	2: 
		WriteFile(
			sNetId := InAmsId,
			hFile := FileHandle,
			pWriteBuff := InPMessage,
			cbWriteLen := InLMessage,
			bExecute := TRUE,
			nErrId => AX_ErrorId[Select],
			bError => AX_Error[Select]
		);
		IF NOT(WriteFile.bBusy) THEN
			IF NOT(WriteFile.bError) THEN
				select := select+1;
				WriteFile(bExecute := FALSE);
				cbWritten := WriteFile.cbWrite;
			ELSE
				select := -1;
			END_IF
		END_IF
	3 : 
		CloseFile(sNetId := InAmsId, 
			hFile := FileHandle,
			bExecute := TRUE, 
			tTimeout := T#1S,
			nErrId => AX_ErrorId[Select],
			bError => AX_Error[Select]
		);
		IF NOT(CloseFile.bBusy) THEN
			IF NOT(CloseFile.bError) THEN
				select := 10;
				CloseFile(bExecute := FALSE);
			ELSE
				select := -1;
			END_IF
		END_IF
		
	10: 
		FileHandle := 0;
		OutBusy := FALSE;
		select := 0;
		OutCompleted := TRUE;
		FOR i := 1 TO NbSteps DO
			AX_ErrorId[i] := 0;
			AX_Error[i] := FALSE;
		END_FOR
		
	-1 : 
		IF FileHandle <> 0 THEN
			CloseFile(sNetId := InAmsId, hFile := FileHandle, bExecute := TRUE);
		END_IF
		OpenFile(bExecute := FALSE);
		WriteFile(bExecute := FALSE);
		IF NOT(CloseFIle.bBusy) THEN
			CloseFile(bExecute := FALSE);
		END_IF
		M_AlarmManager();
		select := 10;
END_CASE

METHOD M_AlarmManager : BOOL
VAR
	j : UINT;
	StringInterm : STRING;
END_VAR
OutError := FALSE;
OutErrorId :='';
FOR j := 1 TO NbSteps DO
	OutError := OutError OR AX_Error[j];
	IF AX_Error[j] THEN
		OutErrorId := concat(concat(Concat(UINT_TO_STRING(j),'_'), UDINT_TO_STRING(AX_ERRORID[j])), CONCAT('*',OutErrorId));
	END_IF
END_FOR
END_METHOD

END_FUNCTION_BLOCK

// ---- 00_FunctionsBlocks/DataProcessing/WriteFile/FUN_CreateDir_CSV.TcPOU
PROGRAM FUN_CreateDir_CSV
VAR_INPUT
	InDirectory 		: T_MaxString;
	Reset2				: BOOL;
END_VAR

VAR
	FB_Time 			: FB_LocalSystemTime;
	MesYear 			: WORD;
	MesMonth			: WORD;
	MesDay				: WORD;
	MesDate				: STRING;
	bTimeOK				: BOOL;
	
	//Dir names 
	CreateDir1			: FB_CreateDir_V2;
	CreateDir2			: FB_CreateDir_V2;
	bFirstDirOk			: BOOL;
	bSecondDirOk		: BOOL;
	bFileOK				: BOOL;
	bDirChange			: BOOL;

END_VAR

VAR_OUTPUT
	
	bInitWrite 			: BOOL;
	AX_DirNames			: ARRAY[1..3] OF t_MaxString; // Folder for years, months and days
	bDirOK				: BOOL;

END_VAR

//	Get time and date  +  Create names
	
IF MesYear <> CalLocalTimeStruct.wYear THEN
	AX_DirNames[1] := Concat(InDirectory, concat(WORD_TO_STRING(CalLocalTimeStruct.wYear), '\'));
	MesYear := CalLocalTimeStruct.wYear;
	bDirChange := TRUE;		
END_IF

IF MesMonth <> CalLocalTimeStruct.wMonth THEN
	AX_DirNames[2] := Concat(AX_DirNames[1], concat(WORD_TO_STRING(CalLocalTimeStruct.wMonth), '\'));
	MesMonth := CalLocalTimeStruct.wMonth;
	bDirChange := TRUE;		
END_IF

IF MesDay <> CalLocalTimeStruct.wDay THEN
	MesDay := CalLocalTimeStruct.wDay;
END_IF		


IF bDirChange OR NOT bFirstDirOk OR NOT bSecondDirOk OR RESET2 THEN
	RESET2 := FALSE;
	bFirstDirOk := FALSE;
	bSecondDirOk := FALSE;
	CreateDir1(InPath := AX_DirNames[1], InExe := TRUE, OutCompleted => bFirstDirOk);
	CreateDir2(InPath := AX_DirNames[2], InExe := bFirstDirOk AND NOT bSecondDirOk, OutCompleted => bSecondDirOk);
	
	IF bFirstDirOk AND bSecondDirOk THEN
		bDirChange := FALSE;
		bDirOK := bFirstDirOk AND bSecondDirOk ;
		CreateDir1(InExe := FALSE);
		CreateDir2(InExe := FALSE);
	END_IF				
END_IF

END_PROGRAM

// ---- 00_FunctionsBlocks/DataProcessing/WriteFile/FB_CreateDir_V2.TcPOU
FUNCTION_BLOCK FB_CreateDir_V2
VAR_INPUT
	InPath 				: T_Maxstring;
	InExe				: BOOL;
END_VAR
VAR_OUTPUT
	OutExiste			: BOOL;
	OutCompleted		: BOOL;
	OutError			: BOOL;
	OutErrorId			: UDINT;
	OutBusy				: BOOL;
END_VAR
VAR
	CreateDir			: FB_CreateDir;	
	
	Trig_Start			: RS;
	Trig				: R_TRIG;
	
	
END_VAR

Trig(CLK := InExe);
//OutCompleted := NOT Trig.Q AND NOT CreateDir.bBusy AND NOT CreateDir.bError;
Trig_Start(SET := Trig.Q);

CreateDir(
	sNetId := '', 
	sPathName := InPath,
	bExecute := Trig.Q
	);
	
IF Trig_Start.Q1 AND NOT CreateDir.bBusy AND (CreateDir.nErrId = 16#723 OR CreateDir.nErrId = 16#70C ) THEN
	createDir(bExecute := FALSE);
	OutExiste := TRUE;
	OutCompleted := TRUE;
	Trig(CLK := FALSE);
	Trig_Start( RESET1 := OutCompleted OR OutError);
	Trig_Start( RESET1 := FALSE);
ELSIF NOT Trig.Q AND Trig_Start.Q1 AND NOT CreateDir.bBusy AND NOT CreateDir.bError THEN
	OutCompleted := TRUE;
	CreateDir(bExecute := FALSE);
	Trig(CLK := FALSE);
	Trig_Start( RESET1 := OutCompleted OR OutError);
	Trig_Start( RESET1 := FALSE);
ELSIF CreateDir.bError THEN
	OutError := TRUE;
	OutErrorId := CreateDir.nErrid;
	CreateDir(bExecute := FALSE);
	Trig(CLK := FALSE);
	Trig_Start( RESET1 := OutCompleted OR OutError);
	Trig_Start( RESET1 := FALSE);

END_IF

OutBusy := Trig_Start.Q1;

END_FUNCTION_BLOCK

// ---- 00_FunctionsBlocks/DataProcessing/ReplaceAll.TcPOU
PROGRAM ReplaceAll
// Replaces all the instances of the input string with another string
// If In_StringToSearch := 'aaaaa123aaaaa123aaaaaaa123aaaaa123'
// In_StringToFind := '123'
// In_StringToReplace : = 'ABC'
// Then : OUT_StringToSearch := 'aaaaaABCaaaaaABCaaaaaaaABCaaaaaABC'
// Equivalent to CTRL + H
VAR_INPUT
	IN_StringToSearch	: T_MaxString;		// String to search : main string with instances we wish to replace
	IN_StringToFind		: STRING;			// String we are looking to find in the String_To_Seach
	IN_StringToReplace 	: STRING;			// String with which we want to replace the String To Find in String To Search
END_VAR

VAR_OUTPUT
	OUT_StringToSearch : T_MaxString;		// Output String
END_VAR

VAR
	KK: INT;
	Test_INT : INT;
END_VAR

OUT_StringToSearch := IN_StringToSearch;
FOR KK := 1 TO LEN(STR := OUT_StringToSearch) DO
	Test_INT := FIND(STR1 := OUT_StringToSearch, STR2 := IN_StringToFind);
	IF Test_INT > 0 THEN
		OUT_StringToSearch := REPLACE(STR1 := OUT_StringToSearch, STR2 := IN_StringToReplace, P := Test_INT, L := len(IN_StringToFind));
		KK := Test_Int;
	END_IF
END_FOR

END_PROGRAM

// ---- 00_FunctionsBlocks/AlarmManagement/FUN_ReadAlarm_CSV.TcPOU
PROGRAM FUN_ReadAlarm_CSV
//Permet de lire les Valeurs de max 1 semaine de points (1 pt/min pdt 7 jours)

VAR_INPUT
	InDirectory_Stockage 		: T_MaxString;		// Base file of the Historization 
	InStartTimeStamp			: TIMESTRUCT;
	InExecute					: BOOL;			//Rising Edge detection of read
	ParamSeparateur				: STRING;
	IN_Reset					: BOOL ; // Close File . 
	ParamMaxLine				: WORD :=  200 ; 
END_VAR                 		

VAR_OUTPUT              		
	OutValue					: ARRAY[1..500] OF ST_ValuesAlarms;
	OutDir						: T_Maxstring;
	OutCompleted				: BOOL;
	OutNbLigne					: UINT;
	OutbBusy					: BOOL;
	OutError 					: BOOL;
	OutErrorID 					: UINT; // 1 : File not found
END_VAR                 		
VAR     
	// Initialisation 
	TypeFile					: STRING;
	ParamTimeOut				: TIME := T#1S;
	
	//Read
	TimeStructBeingRead			: TIMESTRUCT;
	FullDirectory				: STRING;                		
	
	OpenFile					: FB_FileOpen;
	ReadFile					: FB_FileGets;
	CloseFile					: FB_FileClose;
	InfoFile					: FB_EnumFindFileEntry;
	FileInfo					: ST_FindFileEntry;

	Index_Array_OutValue		: UINT := 1;			// Valeur de OutValue qui va être écrite
	
	Opening						: BOOL := TRUE;
	
	LineRead					: T_Maxstring;
	EOF_Reached					: BOOL;              		
	CompteurLigne				: CTU;
	AX_ArrayString 				: ARRAY[1..100] OF T_Maxstring;
	
	OutEmpty					: ARRAY[1..500] OF ST_ValuesAlarms;
	OutBusy						: RS;
	OutCompleted_RS				: RS;
	Trig_Read					: R_TRIG;
	Trig_Start 					: R_TRIG;
	
	FileHandle					: UINT;
	FileHandle_Old				: UINT;
	
	KK: UINT := 1;
	bInit : BOOL;
	LL: UINT;
	MM: UINT;
END_VAR

Trig_Start(CLK := InExecute);
OutCompleted_RS(Reset1 := Trig_Start.Q);
IF trig_start.Q THEN
	OutEmpty := OutValue;
	outError := FALSE;
END_IF
OutBusy(Set := InExecute, RESET1 := OutError OR OutCompleted_RS.Q1);
OutbBusy := OutBusy.Q1;
OutCompleted := OutCompleted_RS.Q1;
IF OutBusy.Q1 THEN	
	// J'initialise le tout : 
	//Initialisation du type de fichier
	TypeFile := 'ALARMS'; 
	
	TimeStructBeingRead := DT_TO_SYSTEMTIME(SYSTEMTIME_TO_DT(InStartTimeStamp) );
	FullDirectory := Concat(Concat(Concat(Concat(Concat(Concat(Concat(Concat(Concat(Concat(Concat(Concat(InDirectory_Stockage , WORD_TO_STRING(TimeStructBeingRead.wyear)),'\'),WORD_TO_STRING(TimeStructBeingRead.wMonth)),'\'),'ALARMS'),'_'),WORD_TO_STRING(TimeStructBeingRead.wyear)),'-'),WORD_TO_STRING(TimeStructBeingRead.wMonth)),'-'),WORD_TO_STRING(TimeStructBeingRead.wDay)),'.csv');
    OutDir := FullDirectory;
	//Ouverture du Fichier, récupération du handle
	OpenFile
	(
		sNetId := '',
		sPathName := FullDirectory,
		nMode := FOPEN_MODEREAD,
		ePath := PATH_GENERIC,
		bExecute := Opening AND NOT OutCompleted_RS.Q1,
		hFile => FileHandle
	);
	
	IF OpenFile.nErrId = 1804 THEN // Le fichier n'existe pas 
		OutErrorID := 1;
		OutError := OpenFile.bError;
		OpenFile(bExecute :=  FALSE);
	ELSIF OpenFile.bError THEN		// Il y a eu une autre erreur
		OutError := OpenFile.bError;
	ELSIF NOT OpenFile.bError AND NOT OpenFile.bBusy AND FileHandle <> 0 AND FileHandle <> FileHandle_Old THEN
		opening := FALSE;
		FileHandle_Old := FileHandle;
	END_IF
	// On a obtenu le file handle, on va commencer la lecture

	// Le bloc suivant va lire le document ligne à ligne en incrémentant le compteur ligne et en ressortant l'ensemble de la ligne dans LineRead
	LineRead := '';
	IF NOT opening THEN
		ReadFile
		(
			sNetId := '',
			hFile := FileHandle,
			bExecute := TRUE,
			tTimeout := ParamTimeOut,
			sLine => LineRead,
			bEOF => EOF_Reached
		);				

		IF NOT ReadFile.bBusy AND NOT ReadFile.bError AND (LineRead <> '') THEN
			ReadFile(bExecute := FALSE);
			CompteurLigne(CU := TRUE);	
			CompteurLigne(CU := FALSE);
			IF CompteurLigne.CV > 2 THEN
				Split(IN_TextToSearch := LineRead, IN_Delimiter := 	ParamSeparateur, OUT_Split => AX_ArrayString);			
				OutValue[Index_Array_OutValue].TimeStamp_Act 	:= AX_ArrayString[1];
				OutValue[Index_Array_OutValue].ID 				:= STRING_TO_UINT(AX_ArrayString[2]);
				OutValue[Index_Array_OutValue].Message			:= AX_ArrayString[3];
				OutValue[Index_Array_OutValue].Value			:= STRING_TO_BOOL(AX_ArrayString[4]);
				OutValue[Index_Array_OutValue].Ack			 	:= STRING_TO_BOOL(AX_ArrayString[5]);
				OutValue[Index_Array_OutValue].Alarms_LVL	 	:= STRING_TO_UINT(AX_ArrayString[6]);				
				Index_Array_OutValue := Index_Array_OutValue + 1;
				
			END_IF
		
		ELSIF NOT ReadFile.bBusy AND  ReadFile.bError THEN
			OutError := TRUE;	
		ELSIF  EOF_Reached THEN
			OutNbLigne := Index_Array_OutValue;
			OutCompleted_RS( SET := TRUE);
			OutCompleted_RS( SET := FALSE);
	
		END_IF	
	
	END_IF
	
ELSIF EOF_Reached AND FileHandle <> 0 THEN
	ReadFile(bExecute := FALSE);
	CloseFile
	(
		sNetId := '',
		bExecute := TRUE,
		hFile := FileHandle,
		tTimeout := ParamTimeOut
	);
	IF NOT CloseFile.bBusy AND NOT CloseFile.bError THEN
		CloseFile(bExecute := FALSE);
		Opening := TRUE;
		CompteurLigne(RESET := TRUE);
		CompteurLigne(RESET := FALSE);
		Index_Array_OutValue := 1;
		FileHandle := 0;
		OutValue := OutEmpty;
	ELSIF NOT CloseFile.bBusy AND closefile.bError THEN
		OutError := TRUE;
	END_IF  
END_IF

END_PROGRAM

// ---- 00_FunctionsBlocks/DataProcessing/Split.TcPOU
PROGRAM Split
//Donne la position de la IN_Position-ième répétition du caractère recherché et renvoie la chaine de caractère suivante
VAR_INPUT
	IN_Delimiter 		: STRING;
	IN_TextToSearch		: T_MaxString;
END_VAR

VAR
	n					: UINT;	
	Position_Int		: UINT;
	LenOutSplit			: INT;
	TextToSearch_Int	: T_MaxString;
	OUT_Null			: ARRAY[1..100] OF T_Maxstring;
END_VAR

VAR_OUTPUT
	OUT_Split			: ARRAY[1..100] OF T_Maxstring;
	NbElements			: UINT;
END_VAR

OUT_Split := OUT_Null;
n:= 1;
TextToSearch_Int := IN_TextToSearch;
Position_Int := INT_TO_UINT( Find(STR1 := TextToSearch_Int, STR2 := IN_Delimiter));
LenOutSplit := 0;

WHILE Position_Int > 0 AND LenOutSplit < LEN(STR:= IN_TextToSearch) DO
	OUT_Split[n] := LEFT(STR := TextToSearch_Int, SIZE := UINT_TO_INT(Position_Int)-1);
	LenOutSplit := LenOutSplit + Len(STR := OUT_Split[n])+1;
	TextToSearch_Int := RIGHT(STR := TextToSearch_Int, SIZE := LEN(STR:= TextToSearch_Int)- LEN(STR:= OUT_Split[n])-1);
	Position_Int := INT_TO_UINT(FIND(STR1 := TextToSearch_Int, STR2 := IN_Delimiter));
	n := n + 1;
END_WHILE

NbElements := n-1;

END_PROGRAM

// ---- 00_FunctionsBlocks/AlarmManagement/SMS_Server.TcPOU
PROGRAM SMS_Server
VAR PERSISTENT
	AX_Numtel						: ARRAY[1..CstNbUser] OF STRING(26) ;	//Contient tous les numéros des utilisateurs
	AX_Subscribed					: ARRAY[1..CstNbUser] OF BOOL ;			//Contient tous les états d'abonnements des utilisateurs aux SMS
	AX_NomUtili						: ARRAY[1..CstNbUser] OF STRING(50);	//Contient tous les noms des utilisateurs
	AX_User_LVL						: ARRAY[1..CstNbUser] OF WORD;			//Contient tous les niveau d'adhésion des utilisateurs.
END_VAR

VAR_INPUT
	IN_DataSetFifo_ReadSMS			: FB_SMSDatasetFifo_Read; //Buffer automate des sms récuperer depuis modem Gsm
	IN_DataSetFifo_SendSMS			: FB_SMSDatasetFifo_Send; //Buffer automate des sms récuperer depuis modem Gsm	
	IN_AX_Journal					: ARRAY [0..CstNbAlarmCode] OF ARRAY[0..15] OF ST_ValuesAlarms; //Journal d'envoi, contient destinataire et message, et gestion de l'envois ou pas du sms
	IN_Reset_OPC					: BOOL;
	IN_ChangePhoneMailInfos_OPC			: BOOL;
	IN_Reset_SmsServer				: BOOL;
	IN_CmdReset_L					: BOOL;
	IN_CmdDeleteAllSms			: BOOL;
END_VAR

VAR
	fbSerialLineControl		: SerialLineControl;
	stTxBufferPC			: ComBuffer;
	stRxBufferPC			: ComBuffer;
	fbReadSMS				: FB_ReadSMS;
	fbSendSMS				: FB_SendSMS;
	fbDeleteSMS				: FB_DeleteSMS;
	fbDeleteAllSMS			: FB_DeleteAllSMS;
	Fblogin 				: FB_Login;
	
	//READ VARIABLE 
	bStartRead				: BOOL; //Gestion du front montant FB ReadSMS
	ReadSMS_bBusy			: BOOL;
	ReadSMS_bError			: BOOL;
	ReadSMS_nErrorID		: UINT;
	
	LoginSMS_bError			: BOOL;
	LoginSMS_bBusy		    : BOOL;
	IndexReadMessage		: USINT:=1; //Index du message a lire
	ReadSMS_MessageText		: STRING(240); // Message brut du SMS recu
	Etape_Read 		 		: SINT:=0; // Etape du Case de M_Fill_Buffer_Read
	Message_Tous_lu 		: BOOL;  // Si tous les message du buffer READ sont lu : True sinon False
	
	//DELETE VARIABLE
	bStartDelete			: BOOL; //Gestion du front montant FB DeleteSms
	DeletedSMS_bBusy		: BOOL;
	DeletedSMS_Error		: BOOL;
	DeletedSMS_nErrorID		: UINT;
	
	IndexDeleteMessage 		: USINT:=1; //Index du message a supprimer
	
	//SEND VARIABLE
	bStartSend				: BOOL;
	Message_Send			: STRING(160);
	MesTimeStamp			: STRING(17);
	SendSMS_bBusy			: BOOL;
	SendSMS_bError			: BOOL;
	Etape_Send				: SINT;
	CPT						: SINT:=1;
	Num_Tel					: STRING(30);

	//INIT VARIABLE
	bStartlogin             : BOOL:=TRUE; //Gestion du front montant FB login
	bInit					: BOOL;
	
	//Variables de All Delete
	DeletedAllSMS_bBusy		: BOOL;
	DeletedAllSMS_Error		: BOOL;
	DeletedAllSMS_nErrorID	: UINT;
	G7_DelAll				: SINT;

	Bstart_delete_all		: BOOL;    
	
	//M_G7_SMS
	CPT_Message				: CTU;
	


	//TABLEAU
	AX_MesAlarmCode_Bool	: ARRAY [1..CstNbAlarmCode] OF ARRAY[1..15] OF BOOL; //Tableau de tous les alarmesCode en Bool
	AX_Alarm_State			: ARRAY [1..CstNbAlarmCode] OF ARRAY[1..15] OF BOOL; //Tableau de Bool avec toutes les nouveaux bit modifiés
	fbXorWord				: FB_XorWord; //Compare 2 Word et retourne les bit modifié
	Extract_Num_Mes			: FB_Extract_Num_Mes; //Extraction des infos: Message,Numero de tel

	// M_Evaluate
	MesDataExd.MesData			: ServerSMS;
	CalNbrUtiliActive    : INT := 10;
	//AlarmCode
	RS_LoginSMS_bError		: RS;
	RS_SendSMS_bError       : RS;
	RS_ReadSMS_bError       : RS;
	RS_DeletedSMS_Error     : RS;
    RS_DeletedAllSMS_Error  : RS;

	AX_Cmd_SMS				: ARRAY[1..CstNbCMD] OF STRING(26):=['Infos','Reboot_ADSL','P_Onduleur','Stop_SMS','Start_SMS','Toggle subscription','Ip Publique','Active Alarms','Help','Test SMS','ForcedStayConnect','Restart HHCollector','Restart PLC','Auto Couplage','Disconnect', 'VPN Connect', 'VPN Disconnect', 'Reboot_IPC']; //Contient toutes les commandes possibles

	Serial_Use				: BOOL:=TRUE;
	ReadAct					: BOOL:=FALSE;
	LoginOK                 : BOOL:=TRUE;
	Reset					: BOOL;
	
	//OPC
	RS_OPC					: RS;
	RS_Deletteall			: RS;
	RS_Reset				: RS;
	Trig_OPC				: R_TRIG;
	Trig_OpcDelAll			: R_TRIG;
	Trig_OpcReset			: R_TRIG;

	
	
END_VAR

IF NOT bInit THEN
	M_Init();
ELSE
	
	// READ OPC Data .
	M_OPC();

	//SERIALLINEMODE_EL6_22B	
	fbSerialLineControl(Mode:= SERIALLINEMODE_PC_COM_PORT ,
		pComIn:= ADR(stPCComInData),
		pComOut:= ADR(stPCComOutData),
		SizeComIn:= UINT_TO_INT( SIZEOF(stPCComInData)),
		TxBuffer:= stTxBufferPC,
		RxBuffer:= stRxBufferPC,
		Error=> ,
		ErrorID=> );
		
	Fblogin(bStart:=bStartlogin ,					// etrangement le login fonctionne puis fait une erreur , puis refonctionne etc . relance du login sur read error je pense qui entraine une tentative de login qui foire. 	
			stTxBuffer:=stTxBufferPC,	
			stRxBuffer:=stRxBufferPC,
			bBusy =>LoginSMS_bBusy,
			bError=>LoginSMS_bError
			);		
		
	fbSendSMS(bStart:= bStartSend,
		sPhoneNumber:= Num_Tel,
		bReset := IN_Reset_OPC ,
		sSMSText:= Message_Send,
		stTxBuffer:=stTxBufferPC ,
		stRxBuffer:=stRxBufferPC,
		bBusy=>SendSMS_bBusy,
		bError=>SendSMS_bError);
	
	fbReadSMS(bStart:= bStartRead,
		nIndex:= IndexReadMessage,
		stTxBuffer:=stTxBufferPC ,
		stRxBuffer:=stRxBufferPC ,
		bBusy=> ReadSMS_bBusy,
		bError=> ReadSMS_bError,
		nErrorID=> ReadSMS_nErrorID
		);
	
	
	fbDeleteSMS
	(
		bStart:= bStartDelete,
		nIndex:= IndexDeleteMessage,
		stTxBuffer:=stTxBufferPC,
		stRxBuffer:=stRxBufferPC,
		bBusy=> DeletedSMS_bBusy,
		bError=> DeletedSMS_Error,
		nErrorID=> DeletedSMS_nErrorID
	);
	
	fbDeleteAllSMS
	(
		bStart:= Bstart_delete_all,
		stTxBuffer:=stTxBufferPC,
		stRxBuffer:=stRxBufferPC,
		bBusy=> DeletedAllSMS_bBusy,
		bError=> DeletedAllSMS_Error,
		nErrorID=> DeletedAllSMS_nErrorID
	);	

	M_DeleteAll();
	M_Fill_Buffer_Read(); //Lecture de tous les messages recu

	M_AlarmManager();
	M_Evaluate();		// Update serveur info
	M_Send(); // Envois de tous les messages (Alarm ou réponce aux sms de cmd)

	M_Cmd_Execute(); // Verification des messages recu
	
	IF Reset OR IN_Reset_OPC  THEN
		M_Reset();
	END_IF
	
	IF NOT LoginSMS_bBusy AND NOT LoginSMS_bError AND LoginOK THEN
		BstartLogin := FALSE;
		Serial_Use:=FALSE;
		LoginOK:=FALSE;
	END_IF
	
	
END_IF

METHOD M_AlarmManager
VAR
	ii:SINT;
	jj:INT;
	KK:INT;
	FB_AlarmCodeManager			: FB_AlarmCodeManager ;
END_VAR
RS_LoginSMS_bError(SET:=LoginSMS_bError,RESET1:=	IN_CmdReset_L OR IN_Reset_OPC); 		
RS_SendSMS_bError(SET:=SendSMS_bError,RESET1:=  	IN_CmdReset_L OR IN_Reset_OPC); 		
RS_ReadSMS_bError(SET:=ReadSMS_bError,RESET1:=  	IN_CmdReset_L OR IN_Reset_OPC); 		
RS_DeletedSMS_Error(SET:=DeletedSMS_Error,RESET1:=	IN_CmdReset_L OR IN_Reset_OPC); 		
RS_DeletedAllSMS_Error(SET:=DeletedAllSMS_Error,RESET1:=IN_CmdReset_L OR IN_Reset_OPC); 	

// ALARM CODE //
	FB_AlarmCodeManager(
		bAlarm1			:= RS_LoginSMS_bErrOR.Q1		  ,			// Login SMS Error
		bAlarm2			:= RS_SendSMS_bErrOR.Q1		   ,			// Send SMS Error
		bAlarm3			:= RS_ReadSMS_bErrOR.Q1		   ,			// Read SMS Error 
		bAlarm4			:= RS_DeletedSMS_ErrOR.Q1		 ,			// Delete SMS Error 
		bAlarm5			:= RS_DeletedAllSMS_ErrOR.Q1	,			// Delete All Sms Error
		bAlarm6			:= IN_DataSetFifo_ReadSMS.bOverwrite,		// Read Fifo overflow
		bAlarm7			:= IN_DataSetFifo_SendSMS.bOverwrite,       // Send Fifo overflow
		bAlarm8			:= FALSE,                                   //
		bAlarm9			:= FALSE,                                   //
		bAlarm10		:= FALSE,                                   //
		bAlarm11		:= FALSE,									//
		bAlarm12		:= FALSE,                                   //
		bAlarm13		:= FALSE,                                   //
		bAlarm14		:= FALSE,                                   //
		bAlarm15		:= FALSE,                                   //
		wAlarmCode		=>MesData.MesAlarmCode);
END_METHOD

METHOD M_Cmd_Execute
VAR_INPUT
END_VAR

VAR
	i: SINT;
	Num_Valide 		: BOOL;
	Message_Valide 	: BOOL;
	Index_CMD 		: SINT;
END_VAR
IF IN_DataSetFifo_ReadSMS.nCount > 0 THEN
	IN_DataSetFifo_ReadSMS.A_Get(); // Récuperation du FIFO
	FOR i:=1 TO CstNbUser DO // VERIFICATION du numéro de telephone
		IF AX_Numtel[i]=IN_DataSetFifo_ReadSMS.Out.Num THEN
			Num_Valide := TRUE;
			EXIT;
		END_IF
	END_FOR
	IF Num_Valide THEN
		FOR i:=1 TO CstNbCMD DO // VERIFICATION du message
			IF IN_DataSetFifo_ReadSMS.Out.Message=AX_Cmd_SMS[i] THEN
				Message_Valide := TRUE;
				Index_CMD:=i;
				EXIT;
			END_IF
		END_FOR
	END_IF
	
	IF Num_Valide AND Message_Valide THEN
		M_G7_SMS(G7_Etape:=Index_CMD);

	ELSE
		IN_DataSetFifo_ReadSMS.A_Remove(); //IL s'agit d'un spam ou d'un utilisateur non autorisé
	END_IF
	

END_IF
END_METHOD

METHOD M_DeleteAll


VAR
	
END_VAR
CASE G7_DelAll OF
	
	0: // Entrée
		IF RS_Deletteall.Q1 AND NOT Serial_Use THEN
			Serial_Use 			:= TRUE;
			Bstart_delete_all 	:= TRUE;
			G7_DelAll 			:= 1;
		END_IF
	1: // attente du bb=usy
		Bstart_delete_all 	:= FALSE;
		IF NOT DeletedAllSMS_bBusy OR DeletedAllSMS_Error THEN
			RS_Deletteall(RESET1:= TRUE);
			RS_Deletteall(RESET1:= FALSE);
			Serial_Use 			:= FALSE;
			G7_DelAll 			:= 0;
		END_IF
		
		
END_CASE
END_METHOD

METHOD M_Evaluate
VAR 
	KK: INT;
END_VAR
CalNbrUtiliActive := 0 ;
FOR KK:=1 TO CstNbUser DO 
	IF 	AX_Numtel[KK] <> '' THEN 
		CalNbrUtiliActive := CalNbrUtiliActive+1 ; 
	END_IF
END_FOR



Mesdata.NbrUtiliActive 	:= CalNbrUtiliActive ;
Mesdata.AX_Numtel		:= AX_Numtel			;
Mesdata.AX_Subscribed	:= AX_subscribed	    ;
MesData.AX_NomUtili		:= AX_NomUtili		    ;
MesData.AX_UserLVL		:= AX_User_LVL		    ;
END_METHOD

METHOD M_Fill_Buffer_Read
CASE Etape_Read OF
	0://Initilisation
		IF NOT ReadSMS_bBusy AND NOT Serial_Use AND ReadAct THEN
			Etape_Read:=10;
			ReadSMS_MessageText:='';
			bStartlogin:=TRUE;
			Serial_Use:=TRUE;
		END_IF
	10: //Initialisation MODEM (ECHO OFF)
		//Serial_Use:=TRUE;
		bStartlogin:=FALSE;
		IF NOT LoginSMS_bBusy AND NOT LoginSMS_bError THEN
			Etape_Read:=1;
			BstartRead:=TRUE;	
		ELSIF LoginSMS_bError THEN
			Etape_Read:=0;
			Serial_Use:=FALSE;
		END_IF
	1://Lecture des sms
		//GVL_Rapale.Serial_Use:=TRUE;
		ReadSMS_MessageText:=fbReadSMS.sMessageText;
		BstartRead:=FALSE;	
		IF NOT ReadSMS_bBusy AND NOT ReadSMS_bError THEN	
			Etape_Read:=2;
			Serial_Use:=FALSE;
		ELSIF ReadSMS_bError THEN
			Etape_Read:=0;
			Serial_Use:=FALSE;
			
		END_IF
		
	2://Analyse du sms en Cas d'un message non vide
		IF(ReadSMS_MessageText<>'OK$R$N') AND (ReadSMS_MessageText<>'') THEN
			
			IF (FIND(ReadSMS_MessageText,'REC UNREAD')>0) THEN		//
				Message_Tous_lu := FALSE;
				IndexReadMessage:=IndexReadMessage+1;
				Extract_Num_Mes(InMessage:=ReadSMS_MessageText);
				IN_DataSetFifo_ReadSMS.A_Add( in := Extract_Num_Mes.OutDataEntry);
				Etape_Read:=0;					
			ELSE	// Messages have already been read. 
				Message_Tous_lu := TRUE;
				IndexReadMessage:=IndexReadMessage+1;
				ReadSMS_MessageText:='';
				Etape_Read:=0;
			END_IF
		ELSE
			Etape_Read:=3;
		END_IF
	3://Analyse du sms en cas de message vide
		IF Message_Tous_lu THEN
			Etape_Read:=4;
		ELSE
			IndexReadMessage:=1;
			Etape_Read:=0;
		END_IF
	4://Initialisation du Delete_FB
		IF NOT DeletedSMS_bBusy AND ReadAct THEN //AND NOT GVL_Rapale.Serial_Use THEN
			Etape_Read:=5;
			bStartDelete:=TRUE;
			Serial_Use:=TRUE;
		END_IF
	5://Suppression du buffer GSM
		//GVL_Rapale.Serial_Use:=TRUE;
			bStartDelete:=FALSE;
		IF NOT DeletedSMS_bBusy AND NOT DeletedSMS_Error THEN
			Serial_Use:=FALSE;
			Etape_Read:=6;
		ELSIF DeletedSMS_Error THEN
			//GVL_Rapale.Serial_Use:=FALSE;
			Etape_Read:=4;
			Serial_Use:=FALSE;
		END_IF
	6://Controle suppression
		IF IndexDeleteMessage=IndexReadMessage-1 THEN
			Etape_Read:=0;
			IndexDeleteMessage:=1;
			Message_Tous_lu:=FALSE;
			IndexReadMessage:=IndexReadMessage+1;
			Serial_Use:=FALSE;
		ELSE
			IndexDeleteMessage:=IndexDeleteMessage+1;
			Etape_Read:=4;
		END_IF		
		
END_CASE
END_METHOD

METHOD M_G7_SMS
VAR_INPUT
	G7_Etape :SINT;
END_VAR

VAR
	InStruct 		: ST_ValuesAlarms;
END_VAR
FUN_Alarms.M_G7_SMS(
	DataSetFifo_ReadSMS		:= IN_DataSetFifo_ReadSMS,
    IN_DataSetFifo_SendSMS	:= IN_DataSetFifo_SendSMS,
 	CPT_Message				:= CPT_Message,	
    InStruct 				:= InStruct,
    G7_Etape 				:= G7_Etape,
    AX_Numtel				:= AX_Numtel,
    AX_subscribed			:= AX_subscribed,
    AX_MesAlarmCode_Bool	:= AX_MesAlarmCode_Bool,
    AX_Cmd_SMS		        := AX_Cmd_SMS
);
END_METHOD

METHOD M_Init

//Initialisation BUFFER

	//Buffer pour la lecture des sms
	IN_DataSetFifo_ReadSMS.A_Reset();
	IN_DataSetFifo_ReadSMS.A_Add();
	IN_DataSetFifo_ReadSMS.A_Get();
	IN_DataSetFifo_ReadSMS.A_Remove();
	
	//Buffer pour l'envois des sms
	IN_DataSetFifo_SendSMS.A_Reset();
	IN_DataSetFifo_SendSMS.A_Add();
	IN_DataSetFifo_SendSMS.A_Get();
	IN_DataSetFifo_SendSMS.A_Remove();

//Initialisation du Journal		
bInit := TRUE;
END_METHOD

METHOD M_OPC : BOOL
VAR
	AX_Numtel_Init				: ARRAY[1..CstNbUser] OF STRING(26);
END_VAR
Trig_OPC(CLK := IN_ChangePhoneMailInfos_OPC);
Trig_OpcDelAll(CLK := IN_CmdDeleteAllSms);
Trig_OpcReset(CLK:= IN_Reset_SmsServer);

RS_OPC(SET:= Trig_OPC.Q);
RS_Deletteall(SET:=Trig_OpcDelAll.Q);
RS_Reset(Set:=Trig_OpcReset.Q);

IF (*NOT Serial_Use AND*) RS_OPC.Q1 THEN
	//Numéro de téléphone
	AX_Numtel := OpcUa.AllValueW.AX_NbPhone_OPC;
	//Nom d'utilisateur
	AX_NomUtili	:= OpcUa.AllValueW.AX_NamesUsers_OPC;
	
	// User LVL . 
	AX_User_LVL := OpcUa.AllValueW.AX_UserLVL;

	//Gestion subscription
	AX_Subscribed := OpcUa.AllValueW.AX_SubscribedSms_OPC;

	RS_OPC(RESET1:= TRUE);
	RS_OPC(Reset1 := FALSE);
END_IF

IF RS_Reset.Q1 THEN
	IN_Reset_Opc := TRUE;
END_IF
END_METHOD

METHOD M_Reset : BOOL
VAR_INPUT
END_VAR
IN_DataSetFifo_SendSMS.A_Reset();

bStartRead 		:= FALSE;
bStartSend 		:= FALSE;
bStartDelete 	:= FALSE;
bStartlogin 	:= FALSE;
Serial_Use		:= FALSE;


SendSMS_Berror := FALSE ;
ReadSMS_bError := FALSE ;
LoginSMS_bError := FALSE ; 
DeletedSMS_Error := FALSE ; 
DeletedAllSMS_Error := FALSE ; 

RS_Reset(RESET1 := TRUE);
RS_Reset(RESET1 := FALSE);
Reset 			:= FALSE;
IN_Reset_OPC 		:= FALSE;
END_METHOD

METHOD M_Send
VAR_INPUT
END_VAR

CASE ETAPE_Send OF
	0://Etape d'entree
		IF NOT SendSMS_bBusy  AND NOT Serial_Use AND IN_DataSetFifo_SendSMS.nCount > 0 AND NOT LoginSMS_bBusy AND NOT LoginSMS_bError THEN  //Si serial libre et buffer contient plus d'une infos
			ReadAct:=FALSE;	
			Serial_Use:=TRUE;
			//bStartSend:=TRUE;
			SendSMS_bError := FALSE;
			Num_Tel := '';
			Message_Send:='';
			IN_DataSetFifo_SendSMS.A_Get();  //recuperation du message dans le send buffer 
			ETAPE_Send := 20  ; 
		ELSE
			ReadAct:=TRUE;	// En attente de lecture de mot d'alarme
		END_IF
			
		20:// Check les utilisateurs pour l'envoi des SMS 
			IF AX_Numtel[CPT] <> '' AND  AX_Subscribed[CPT] AND IN_DataSetFifo_SendSMS.out.Num_tel = '' AND (AX_User_LVL[CPT] AND IN_DataSetFifo_SendSMS.out.Alarms_LVL)>0    THEN
				// On envoi l'alarme si l'utilisateur est subscribed , et est dans la liste de diffusion de l'alarme
				Num_Tel:=AX_NumTel[CPT];
				bStartSend:=TRUE;
				ETAPE_Send:=1;
				MesTimeStamp := CONCAT(REPLACE(STR1:= IN_DataSetFifo_SendSMS.Out.TimeStamp_Act, STR2 := ' ', L := 1, P := 11), ' ') ;

				Message_Send := CONCAT(str1:=CONCAT(str1:=CONCAT(str1:=MesTimeStamp, str2:='$NID:' ), STR2:= UINT_TO_STRING(IN_DataSetFifo_SendSMS.out.ID)), STR2:=' ,' ) ; 
				Message_Send := CONCAT(STR1:=Message_Send , STR2:= IN_AX_Journal[IN_DataSetFifo_SendSMS.out.IndexWord][IN_DataSetFifo_SendSMS.Out.IndexBit].Message);
				
				IF IN_DataSetFifo_SendSMS.OUT.Active  THEN //Connaitre le statut de l'alarme: Active ou Non active
					Message_Send:=Concat(left(Message_Send, 125),' : Active');	// ajout de la mention activee ou desactive 
				ELSE
					Message_Send:=concat(left(Message_Send, 125),' : Desactive');
				END_IF
			ELSIF ( NOT AX_Subscribed[CPT] OR (AX_User_LVL[CPT] AND IN_DataSetFifo_SendSMS.out.Alarms_LVL)=0  ) AND IN_DataSetFifo_SendSMS.out.Num_tel = ''  THEN
				// L'alarme n'est pas envoyéeà cet utilisateur	
				Num_Tel := '';
				ETAPE_Send:=2;
			ELSIF IN_DataSetFifo_SendSMS.out.Num_tel <> ''  THEN
				// Si un numero de telephone est renseigné précisement, on envoi à ce numéro quelque soit la liste de diffusion , ou si l'utilisateur est subscribed
				bStartSend:=TRUE;
				Message_Send := CONCAT(STR1:=Message_Send , STR2:= IN_AX_Journal[IN_DataSetFifo_SendSMS.out.IndexWord][IN_DataSetFifo_SendSMS.Out.IndexBit].Message);
				Num_Tel:=IN_DataSetFifo_SendSMS.Out.Num_tel;
				ETAPE_Send:=1;
			ELSE
				// L'alarme n'est pas envoyée		
				Num_Tel := '';
				ETAPE_Send:=2;
			END_IF

	1://Envois du message
		Bstartsend:=FALSE;	
		IF NOT SendSMS_bBusy  THEN
			IF IN_DataSetFifo_SendSMS.OUT.IndexWord > 0 AND IN_DataSetFifo_SendSMS.In.Num_tel = ''   THEN
				ETAPE_Send:=2; // Alarme
				
			ELSE
				ETAPE_Send:=3; // Retour Sms ou utilisateur de renseignée
			END_IF
		ELSIF NOT SendSMS_bBusy AND SendSMS_Berror THEN // GGY
			//ETAPE_Send:=0; modif lWN seminaire 26/08/2020, gestion des ATE0, si erreur on supprime tout de meme le sms.
			ETAPE_Send:= 3;
			SendSMS_Berror := FALSE ; // On reset l'error apres avoir supprimé le SMS . 
			
		END_IF
		
	2:// Switch a un autre utilisateur
		IF CPT< CstNbUser THEN
			CPT:=CPT+1;
			ETAPE_Send:=20;
		ELSE
			ETAPE_Send:=3;
		END_IF
	
	3://Suppression de l'alarme et on passe au prochaine element dans le fifo
		IN_DataSetFifo_SendSMS.A_Remove();
		CPT:=1;
		Message_Send:='';
		ETAPE_Send:=0;
		Serial_Use:=FALSE;
		bStartSend:=FALSE;

END_CASE
END_METHOD

END_PROGRAM

// ---- 00_FunctionsBlocks/Fifo/FB_SMSDatasetFifo_Read.TcPOU
FUNCTION_BLOCK FB_SMSDatasetFifo_Read
VAR_INPUT
    bOverwrite : BOOL;
    In         : ST_SMSDataSetEntry_Read;
END_VAR
VAR_OUTPUT
    bOk        : BOOL;
    nCount     : UDINT;
    nLoad      : UDINT;
    Out        : ST_SMSDataSetEntry_Read;
END_VAR
VAR
    arrBuffer  : ARRAY[0..Max_buffer_size_G] OF BYTE; (* Buffer memory used by FB_MemRingBuffer function block *)
    fbBuffer   : FB_MemRingBuffer;
END_VAR

ACTION A_Add:
fbBuffer.A_AddTail(pWrite := ADR(in),
						   cbWrite:=SIZEOF(in),
						   pBuffer:=ADR(arrBuffer),
						   cbBuffer:=SIZEOF(arrBuffer),
						   bOK=>bOK,
						   nCount =>nCount);
IF NOT bOK THEN 
	IF bOverwrite THEN
		fbBuffer.A_RemoveHead();(*remove one oldest entry*)
		fbBuffer.A_AddTail(bOK => bOk,nCount => nCount);
	END_IF
END_IF

nload := (fbbuffer.cbSize * 100)/(Max_buffer_size_G);
END_ACTION

ACTION A_Get:
fbBuffer.A_GetHead(pWrite := ADR(out),
						   cbWrite:=SIZEOF(out),
						   pBuffer:=ADR(arrBuffer),
						   cbBuffer:=SIZEOF(arrBuffer),
						   bOK=>bOK,
						   nCount =>nCount);
nload := (fbbuffer.cbSize * 100)/(Max_buffer_size_G);
END_ACTION

ACTION A_Remove:
fbBuffer.A_RemoveHead(pRead:=ADR(out),
						cbRead:=SIZEOF(out),
						pBuffer:=ADR(arrBuffer),
						cbBuffer:=SIZEOF(arrBuffer),
						bOK=>bOK,
						nCount =>nCount);
nload := (fbbuffer.cbSize * 100)/(Max_buffer_size_G);
END_ACTION

ACTION A_Reset:
MEMSET(ADR(arrBuffer),0,SIZEOF(arrBuffer)); (*reset internal buffer*)
fbBuffer.A_Reset(bOK=>bOK,nCount=>ncount);
nload := (fbbuffer.cbSize * 100)/(Max_buffer_size_G);
END_ACTION

END_FUNCTION_BLOCK

// ---- 00_FunctionsBlocks/Fifo/FB_SMSDatasetFifo_Send.TcPOU
FUNCTION_BLOCK FB_SMSDatasetFifo_Send
VAR_INPUT
    bOverwrite : BOOL;
    In         : ST_SMSDataSetEntry_Send;
END_VAR
VAR_OUTPUT
    bOk        : BOOL;
    nCount     : UDINT;
    nLoad      : UDINT;
    Out        : ST_SMSDataSetEntry_Send;
END_VAR
VAR
    arrBuffer  : ARRAY[0..Max_buffer_size_G] OF BYTE; (* Buffer memory used by FB_MemRingBuffer function block *)
    fbBuffer   : FB_MemRingBuffer;
END_VAR

ACTION A_Add:
fbBuffer.A_AddTail(pWrite := ADR(in),
						   cbWrite:=SIZEOF(in),
						   pBuffer:=ADR(arrBuffer),
						   cbBuffer:=SIZEOF(arrBuffer),
						   bOK=>bOK,
						   nCount =>nCount);
IF NOT bOK THEN 
	IF bOverwrite THEN
		fbBuffer.A_RemoveHead();(*remove one oldest entry*)
		fbBuffer.A_AddTail(bOK => bOk,nCount => nCount);
	END_IF
END_IF

nload := (fbbuffer.cbSize * 100)/(Max_buffer_size_G);
END_ACTION

ACTION A_Get:
fbBuffer.A_GetHead(pWrite := ADR(out),
						   cbWrite:=SIZEOF(out),
						   pBuffer:=ADR(arrBuffer),
						   cbBuffer:=SIZEOF(arrBuffer),
						   bOK=>bOK,
						   nCount =>nCount);
nload := (fbbuffer.cbSize * 100)/(Max_buffer_size_G);
END_ACTION

ACTION A_Remove:
fbBuffer.A_RemoveHead(pRead:=ADR(out),
						cbRead:=SIZEOF(out),
						pBuffer:=ADR(arrBuffer),
						cbBuffer:=SIZEOF(arrBuffer),
						bOK=>bOK,
						nCount =>nCount);
nload := (fbbuffer.cbSize * 100)/(Max_buffer_size_G);
END_ACTION

ACTION A_Reset:
MEMSET(ADR(arrBuffer),0,SIZEOF(arrBuffer)); (*reset internal buffer*)
fbBuffer.A_Reset(bOK=>bOK,nCount=>ncount);
nload := (fbbuffer.cbSize * 100)/(Max_buffer_size_G);
END_ACTION

END_FUNCTION_BLOCK

// ---- 00_FunctionsBlocks/Communication/SMS/FB_ReadSMS.TcPOU
FUNCTION_BLOCK FB_ReadSMS

VAR_INPUT PERSISTENT 
	ParamTimeoutReadSMS		: TIME := T#3S ; // Tiemout pour lire les sms.  Attention , ce parametre est très important . Si pas assez grand, risque de données tronquées. 
	
	
	
END_VAR

VAR_INPUT
	bStart					: BOOL;
	nIndex					: USINT;
	
END_VAR
VAR_OUTPUT
	sMessageText			: STRING(240);
	bBusy					: BOOL;
	bError					: BOOL;
	nErrorID				: UINT;
	
END_VAR

VAR_IN_OUT
	stTxBuffer				: ComBuffer;
	stRxBuffer				: ComBuffer;
END_VAR

VAR
	rtrigStart				: R_TRIG;

	fbSendData				: SendData;
	fbReceiveData			: ReceiveData;
	fbClearComBuffer		: ClearComBuffer;

	i,iSavedIndex			: INT;
	uiAnalyzeAnswer			: UINT;
	nStep					: UINT; (* sequence state *)
	tonWaitTime				: TON;
	tonTimeOut				: TON;
	tTimeout				: TIME:=T#30S;


	arAnswerOK				: ARRAY[1..2] OF BYTE:=[16#4F,16#4B];
	arAnswerErr				: ARRAY[1..5] OF BYTE:=[16#45,16#52,16#52,16#4F,16#52];

	sReadSMS				: STRING(15);			(*Command-String*)
	arReadSMS				: ARRAY[1..15] OF BYTE; (*Command-ARRAY*)
	arReadSMSAnswerRcv		: ARRAY[1..300] OF BYTE;(*Received answer of the command*)
	arReadSMSAnswerClr		: ARRAY[1..300] OF BYTE;(*Empty-ARRAY to clear the answer for debugging*)
END_VAR


	rtrigStart(CLK:=bStart);

	tonTimeout();
	IF (tonTimeout.Q) THEN
		tonTimeout(IN := FALSE);
		nStep := 900;
	END_IF


	CASE nStep OF

	0: 	(*Idle Step*);
		MEMSET(ADR(sMessageText),0,SIZEOF(sMessageText));
		tonTimeout(IN:=FALSE);
		IF (rtrigStart.Q AND NOT bBusy) THEN
			nStep := 5;
			bBusy := TRUE;
			
		ELSE
			bBusy := FALSE;
		END_IF


	5:
		bError					:= FALSE;
		nErrorId				:= 0;
		tonWaitTime				(IN := FALSE);
		tonTimeout				(IN := TRUE, PT := tTimeout);
		fbClearComBuffer		(buffer:=stRxBuffer);
		fbClearComBuffer		(buffer:=stTxBuffer);
		sMessageText			:= '';
		MEMSET(ADR(sMessageText),0,SIZEOF(sMessageText));
		nStep := 50;


	50:(*Create command-Arrays*)
		(*Read SMS*)
		sReadSMS:='AT+CMGR="';
		sReadSMS:=CONCAT(sReadSMS,USINT_TO_STRING(nIndex));
		sReadSMS:=CONCAT(sReadSMS,'"X');	(*The "X" is a placeholder in the send-string
											for the "CR" (Hex 0D) in the send-Array*)
		MEMCPY(ADR(arReadSMS),ADR(sReadSMS),LEN(sReadSMS)); (*Copy String to ARRAY*)
		arReadSMS[LEN(sReadSMS)]:=16#0D;	(*Place the "CR" in the array*)

		nStep	:= 100;


	100:(*Send read-command*)
		fbSendData(
		pSendData:=ADR(arReadSMS),
		Length:= LEN(sReadSMS),
		TXbuffer:= stTxBuffer);

		IF NOT fbSendData.Busy THEN
			nStep:=110;
		END_IF

		IF  fbSendData.Error<>0 THEN
			bError:= TRUE;
			nErrorID:= fbSendData.Error;
			nStep:=1000;
		END_IF


	110:(*The beginning and the contents of the answer can vary. If the message-slot contains
		a valid message	it begins with "+CMGR" and ends with "OK". 
		An answer of an empty slot is only "OK". In case of an error the answer is only "ERROR"
		So there is no proper prefix to wait fOR *)
		fbReceiveData(
		pPrefix:= 0,
		LenPrefix:= 0,
		pReceiveData:= ADR(arReadSMSAnswerRcv),
		SizeReceiveData:= SIZEOF(arReadSMSAnswerRcv),
		Timeout:= ParamTimeoutReadSMS ,		
		RXbuffer:= stRxBuffer);

		(*Telegram is received*)
		IF 			fbReceiveData.DataReceived
			AND NOT fbReceiveData.busy	THEN
						nStep:=120;
		END_IF


	120:(* NEW VERSION  : ON recupère la commande si elle est non vide ou non pleine. on analyze les champs ensuite.*)

		(* OLD VERSION  : Find an "OK" or an "ERROR"-Part in the answer
		Search from the end of the received string to the top and take the first match
		not to get a SMS-written "ok" or "error"*)
		uiAnalyzeAnswer	:=0;
		iSavedIndex		:=0;
		IF arReadSMSAnswerRcv[SIZEOF(arReadSMSAnswerRcv)]<> 0 THEN		
			nErrorID := 16#FFFF; // La taille du message dépasse ce que l'on peut récupérer
		ELSIF arReadSMSAnswerRcv[1]= 0 THEN 
			nErrorID := 16#800E; // Le message est vide 
		ELSE
			
			FOR i:= UINT_TO_INT(SIZEOF(arReadSMSAnswerRcv)) TO 1 BY -1 DO		// i:= uint_to_int(SIZEOF(arReadSMSAnswerRcv)-5) TO 1 BY -1 DO	
				IF 		arReadSMSAnswerRcv[i]	<> 0 THEN 	//= arAnswerOK[1] AND arReadSMSAnswerRcv[i+1] 	= arAnswerOK[2]		THEN
						
						iSavedIndex:=i;// iSavedIndex:=i-1;
						
						IF iSavedIndex > 2 THEN 
							uiAnalyzeAnswer:=1;		(*Read SMS successfully executed*)
						ELSE
							uiAnalyzeAnswer:=0;		(*Read SMS successfully executed*)
							nErrorID := 16#FFFF; // La taille du message est inférieru à deux word , on ne peut pas le copier dans un string
						END_IF
						
					EXIT;
	(*
				ELSIF	arReadSMSAnswerRcv[i]		= arAnswerErr[1]
					AND arReadSMSAnswerRcv[i+1] 	= arAnswerErr[2]
					AND arReadSMSAnswerRcv[i+2] 	= arAnswerErr[3]
					AND arReadSMSAnswerRcv[i+3] 	= arAnswerErr[4]
					AND arReadSMSAnswerRcv[i+4] 	= arAnswerErr[5]	THEN
						uiAnalyzeAnswer:=2;		(*Read SMS failed*)
					EXIT;
					*)
				END_IF
			END_FOR
			
		END_IF
		CASE uiAnalyzeAnswer OF
			0:(*Undefined Answer*)
				bError:= TRUE;
				//nErrorID:= 16#800E;
				nStep:=1000;
				//nStep:=1000;

			1:(*Read SMS successfully executed*)
				nStep:=130;

			2:(*Read SMS failed*)
				bError:= TRUE;
				nErrorID:= 16#800D;
				nStep:=1000;
		END_CASE


	130:(*Copy message-Array to String*)
		MEMCPY(ADR(sMessageText),(ADR(arReadSMSAnswerRcv)+2),(iSavedIndex)); (*"2" : Do not read the first two digits of the answer. It always begins with "0D,0A"*)

		IF (FIND(sMessageText,'ERROR')>0) THEN 
			// Il y a une erreru dans la lecture du message. 
			bError := TRUE ; 
			nErrorID:= 16#800D;
			nStep:=1000;
		ELSE 
			nStep:=1000;
		END_IF



	900:(*Timeout*)
		bError:= TRUE;
		nErrorID:= 16#8001;
		nStep:=1000;


	1000:(*Reset Receive-FB*)
		fbReceiveData(	Reset:=TRUE,RXbuffer:= stRxBuffer);
		tonWaitTime(IN:=TRUE, PT:=t#500ms);
		IF	tonWaitTime.Q	THEN
			fbReceiveData(	Reset:=FALSE,RXbuffer:= stRxBuffer);
			nStep:=1010;
		END_IF


	1010:(*Send/Receive successful -> Reset FBs*)
		fbClearComBuffer(buffer:=stRxBuffer);
		fbClearComBuffer(buffer:=stTxBuffer);
		arReadSMSAnswerRcv	:= arReadSMSAnswerClr;
		nStep:=0;
		bBusy:=FALSE;

	END_CASE;

END_FUNCTION_BLOCK

// ---- 00_FunctionsBlocks/Communication/SMS/FB_SendSMS.TcPOU
FUNCTION_BLOCK FB_SendSMS

VAR_INPUT
	bStart					: BOOL;  			(* Rising edge start fb execution *)
	sPhoneNumber			: STRING(30);		(* phone Number *)
	sSMSText				: T_MaxString;		(* Message Text *)
	bReset					: BOOL ; 
END_VAR

VAR_OUTPUT
	bBusy					: BOOL;
	bError					: BOOL;
	nErrorID				: UINT;
	
END_VAR

VAR_IN_OUT
	stTxBuffer				: ComBuffer;
	stRxBuffer				: ComBuffer;
	
END_VAR

VAR
	rtrigStart				: R_TRIG;

	fbSendData				: SendData;
	fbReceiveData			: ReceiveData;
	fbClearComBuffer		: ClearComBuffer;

	i						: UINT;
	uiAnalyzeAnswer			: UINT;
	nStep					: UINT; (* sequence state *)
	tonWaitTime				: TON;
	tonTimeOut				: TON;
	tTimeout				: TIME:=T#60S;

	byAnswerEnter			: BYTE:=16#3E; //">"
	arAnswerCMGS			: ARRAY[1..4] OF BYTE:=[16#43,16#4D,16#47,16#53]; //CMGS
	arAnswerOK				: ARRAY[1..2] OF BYTE:=[16#4F,16#4B]; //OK
	arAnswerErr				: ARRAY[1..5] OF BYTE:=[16#45,16#52,16#52,16#4F,16#52]; //ERROR

	sSetSMSFormat			: STRING(10);			(*Command-String*)
	arSetSMSFormat			: ARRAY[1..10] OF BYTE;	(*Command-ARRAY*)
	arSetSMSFormatAnswerRcv	: ARRAY[1..5] OF BYTE;	(*Received answer of the command*)
	arSetSMSFormatAnswerClr	: ARRAY[1..5] OF BYTE;	(*Empty-ARRAY to clear the answer for debugging*)

	sSendSMSPart1			: STRING(40);			(*Command-String*)
	arSendSMSPart1			: ARRAY[1..40] OF BYTE;	(*Command-ARRAY*)
	arSendSMSPart1AnswerRcv	: ARRAY[1..5] OF BYTE;	(*Received answer of the command*)
	arSendSMSPart1AnswerClr	: ARRAY[1..5] OF BYTE;	(*Empty-ARRAY to clear the answer for debugging*)

	sSendSMSPart2			: STRING(170);			(*Command-String*)
	arSendSMSPart2			: ARRAY[1..170] OF BYTE;(*Command-ARRAY*)
	arSendSMSPart2AnswerRcv	: ARRAY[1..35] OF BYTE;	(*Received answer of the command*)
	arSendSMSPart2AnswerClr	: ARRAY[1..35] OF BYTE;	(*Empty-ARRAY to clear the answer for debugging*)
END_VAR


IF bReset THEN 
	bError := FALSE ; 
	bReset:= FALSE ; 
END_IF


	rtrigStart(CLK:=bStart);

	tonTimeout();
	IF (tonTimeout.Q) THEN
		tonTimeout(IN := FALSE);
		nStep := 900;
	END_IF


	CASE nStep OF

	0:	(*Idle Step*);
		tonTimeout(IN:=FALSE);
		IF (rtrigStart.Q AND NOT bBusy) THEN
			nStep := 5;
			bBusy := TRUE;
		ELSE
			bBusy := FALSE;
		END_IF


	5:
		bError					:= FALSE;
		nErrorId				:= 0;
		tonWaitTime				(IN := FALSE);
		tonTimeout				(IN := TRUE, PT := tTimeout);
		fbClearComBuffer		(buffer:=stRxBuffer);
		fbClearComBuffer		(buffer:=stTxBuffer);
		arSetSMSFormatAnswerRcv	:= arSetSMSFormatAnswerClr;
		arSendSMSPart1AnswerRcv	:= arSendSMSPart1AnswerClr;
		arSendSMSPart2AnswerRcv	:= arSendSMSPart2AnswerClr;
	
		nStep := 10;


	10:(*Length of phone-number within limits?*)
		IF 		LEN(sPhoneNumber) < 1
			OR	LEN(sPhoneNumber) > 25 THEN
			bError		:= TRUE;
			nErrorID	:= 16#8006;
			nStep		:= 1000;
		ELSE
			nStep		:= 20;
		END_IF


	20:(*Phone-number contains correct characters? 0..9, + *)
		FOR i:=1 TO LEN(sPhoneNumber) DO
			IF 	((ASC(MID(sPhoneNumber,1,i)) < 16#30) OR (ASC(MID(sPhoneNumber,1,i)) > 16#39))
				AND NOT (ASC(MID(sPhoneNumber,1,i)) = 16#2B)	THEN
				bError		:= TRUE;	(*a non-numeric character in the phone-number, except the "+"-sign*)
				nErrorID	:= 16#8007;
			END_IF
		END_FOR

		IF bError	THEN
			nStep	:= 1000;
		ELSE
			nStep	:= 30;
		END_IF


	30:(*Length of SMS-Text within limits?*)
		IF 	(LEN(sSMSText) < 1 OR LEN(sSMSText) > 160) THEN
			bError		:= TRUE;
			nErrorID	:= 16#8008;
			nStep		:= 1000;
		ELSE
			nStep		:= 50;
		END_IF


	50:(*Create command-Arrays*)

		(*Set SMS Format to textmode*)
		sSetSMSFormat:='AT+CMGF=1';
		sSetSMSFormat:=CONCAT(sSetSMSFormat,'X');	(*The "X" is a placeholder in the send-string
													for the "CR" (Hex 0D) in the send-Array*)
		MEMCPY(ADR(arSetSMSFormat),ADR(sSetSMSFormat),LEN(sSetSMSFormat)); (*Copy String to ARRAY*)
		arSetSMSFormat[LEN(sSetSMSFormat)]:=16#0D;	(*Place the "CR" in the array*)


		(*Send SMS, Part1 - Phone-number*)
		sSendSMSPart1:='AT+CMGS="';
		sSendSMSPart1:=CONCAT(sSendSMSPart1,sPhoneNumber);
		sSendSMSPart1:=CONCAT(sSendSMSPart1,'"X');	(*The "X" is a placeholder in the send-string
													for the "CR" (Hex 0D) in the send-Array*)
		MEMCPY(ADR(arSendSMSPart1),ADR(sSendSMSPart1),LEN(sSendSMSPart1)); (*Copy String to ARRAY*)
		arSendSMSPart1[LEN(sSendSMSPart1)]:=16#0D;	(*Place the "CR" in the array*)


		(*Send SMS, Part2 - text*)
		sSendSMSPart2:='"';
		sSendSMSPart2:=CONCAT(sSendSMSPart2,sSMSText);
		sSendSMSPart2:=CONCAT(sSendSMSPart2,'"X');	(*The "X" is a placeholder in the send-string
													for the "ctrl+z" (Hex 1A) in the send-Array*)
		MEMCPY(ADR(arSendSMSPart2),ADR(sSendSMSPart2),LEN(sSendSMSPart2)); (*Copy String to ARRAY*)
		arSendSMSPart2[LEN(sSendSMSPart2)]:=16#1A;	(*Place the "ctrl+z" in the array*)


		nStep	:= 100;


	100:(*Set SMS-Format to text-Mode*)
		fbSendData(
		pSendData:=ADR(arSetSMSFormat),
		Length:= LEN(sSetSMSFormat),
		TXbuffer:= stTxBuffer);

		IF NOT fbSendData.Busy THEN
			nStep:=110;
		END_IF

		IF  fbSendData.Error<>0 THEN
			bError:= TRUE;
			nErrorID:= fbSendData.Error;
			nStep:=1000;
		END_IF


	110:(*Wait for OK or Err-Answer. Any other answer caused by Comm-Error will end in global timeout*)
		fbReceiveData(
		pPrefix:= 0,
		LenPrefix:= 0,
		pReceiveData:= ADR(arSetSMSFormatAnswerRcv),
		SizeReceiveData:= SIZEOF(arSetSMSFormatAnswerRcv),
		Timeout:= t#500ms,
		RXbuffer:= stRxBuffer);

		(*Telegram is received*)
		IF 			fbReceiveData.DataReceived
			AND NOT fbReceiveData.busy	THEN
						nStep:=120;
		END_IF


	120:(*Analyze answer*)
		IF		(arSetSMSFormatAnswerRcv[3]=arAnswerOK[1]) AND (arSetSMSFormatAnswerRcv[4]=arAnswerOK[2])	THEN
					nStep:=200;			(*Set-format successfully executed*)
		ELSIF	(arSetSMSFormatAnswerRcv[3]=arAnswerErr[1]) AND (arSetSMSFormatAnswerRcv[4]=arAnswerErr[2])	THEN
					bError:= TRUE;
					nErrorID:= 16#8009;	(*Set-format failed*)
					nStep:=1000;
		ELSE
					bError:= TRUE;
					nErrorID:= 16#800A;	(*Undefined answer*)
					nStep:=1000;
		END_IF


	200:(*Send SMS Part1 - Command and phone-number*)
		fbSendData(
		pSendData:=ADR(arSendSMSPart1),
		Length:= LEN(sSendSMSPart1),
		TXbuffer:= stTxBuffer);

		IF NOT fbSendData.Busy THEN
			nStep:=210;
		END_IF

		IF  fbSendData.Error<>0 THEN
			bError:= TRUE;
			nErrorID:= fbSendData.Error;
			nStep:=1000;
		END_IF


	210:(*Wait explicitly for an ">"-Answer because normally only ">" is possible,
		any other answer is regarded faulty and will end in global timeout*)

		fbReceiveData(
		pPrefix:= ADR(byAnswerEnter),
		LenPrefix:= 1,
		pReceiveData:= ADR(arSendSMSPart1AnswerRcv),
		SizeReceiveData:= SIZEOF(arSendSMSPart1AnswerRcv),
		Timeout:= t#500ms,
		Reset:= FALSE,
		RXbuffer:= stRxBuffer);

		(*Telegram is received*)
		IF 			fbReceiveData.DataReceived
			AND NOT fbReceiveData.busy			THEN
						nStep:=220;
		END_IF


	220:(*Send SMS Part2 - text-part*)
		fbSendData(
		pSendData:=ADR(arSendSMSPart2),
		Length:= LEN(sSendSMSPart2),
		TXbuffer:= stTxBuffer);

		IF NOT fbSendData.Busy THEN
			nStep:=230;
		END_IF

		IF  fbSendData.Error<>0 THEN
			bError:= TRUE;
			nErrorID:= fbSendData.Error;
			nStep:=1000;
		END_IF


	230:(*Wait explicitly for a "CMGS"-Answer because normally only "CMGS" is possible,
		any other answer is regarded faulty and will end in global timeout*)
		fbReceiveData(
		pPrefix:= ADR(arAnswerCMGS),
		LenPrefix:= SIZEOF(arAnswerCMGS),
		pReceiveData:= ADR(arSendSMSPart2AnswerRcv),
		SizeReceiveData:= SIZEOF(arSendSMSPart2AnswerRcv),
		Timeout:= t#1000ms,
		RXbuffer:= stRxBuffer);

		(*Telegram is received*)
		IF 			fbReceiveData.DataReceived
			AND NOT fbReceiveData.busy	THEN
						nStep:=240;
		END_IF


	240:(*Find an "OK" or an "ERROR"-Part in the answer*)
		uiAnalyzeAnswer:=0;
		FOR i:= 1 TO (SIZEOF(arSendSMSPart2AnswerRcv)-5) DO
			IF 		arSendSMSPart2AnswerRcv[i]		= arAnswerOK[1]
				AND arSendSMSPart2AnswerRcv[i+1] 	= arAnswerOK[2]		THEN
					uiAnalyzeAnswer:=1;		(*Send SMS successfully executed*)
					EXIT;

			ELSIF	arSendSMSPart2AnswerRcv[i]		= arAnswerErr[1]
				AND arSendSMSPart2AnswerRcv[i+1] 	= arAnswerErr[2]
				AND arSendSMSPart2AnswerRcv[i+2] 	= arAnswerErr[3]
				AND arSendSMSPart2AnswerRcv[i+3] 	= arAnswerErr[4]
				AND arSendSMSPart2AnswerRcv[i+4] 	= arAnswerErr[5]	THEN
					uiAnalyzeAnswer:=2;		(*Send SMS failed*)
					EXIT;
			END_IF
		END_FOR

		CASE uiAnalyzeAnswer OF
			0:(*Undefined Answer*)
				bError:= TRUE;
				nErrorID:= 16#800D;
				nStep:=1000;

			1:(*Send SMS successfully executed*)
				nStep:=1000;

			2:(*Send SMS failed*)
				bError:= TRUE;
				nErrorID:= 16#800C;
				nStep:=1000;
		END_CASE


	900:(*Timeout*) // delete last sms in case of timeout
		bError:= TRUE;
		nErrorID:= 16#8001;
		nStep:=1000;


	1000:(*Reset Receive-FB*)
		fbReceiveData(	Reset:=TRUE,RXbuffer:= stRxBuffer);
		tonWaitTime(IN:=TRUE, PT:=t#500ms);
		IF	tonWaitTime.Q	THEN
			fbReceiveData(	Reset:=FALSE,RXbuffer:= stRxBuffer);
			nStep:=1010;
		END_IF


	1010:	(*Send/Receive successful -> Reset FBs*)
		fbClearComBuffer(buffer:=stRxBuffer);
		fbClearComBuffer(buffer:=stTxBuffer);
		nStep:=0;
		bBusy:=FALSE;

	END_CASE;

END_FUNCTION_BLOCK

// ---- 00_FunctionsBlocks/Communication/SMS/FB_DeleteSMS.TcPOU
FUNCTION_BLOCK FB_DeleteSMS
VAR_INPUT
	bStart					: BOOL;
	nIndex					: USINT;
END_VAR
VAR_OUTPUT
	bBusy					: BOOL;
	bError					: BOOL;
	nErrorID				: UINT;
END_VAR

VAR_IN_OUT
	stTxBuffer				: ComBuffer;
	stRxBuffer				: ComBuffer;
END_VAR

VAR
	rtrigStart				: R_TRIG;

	fbSendData				: SendData;
	fbReceiveData			: ReceiveData;
	fbClearComBuffer		: ClearComBuffer;

	i						: INT;
	uiAnalyzeAnswer			: UINT;
	nStep					: UINT; (* sequence state *)
	tonWaitTime				: TON;
	tonTimeOut				: TON;
	tTimeout				: TIME:=t#5s;

	arAnswerOK				: ARRAY[1..2] OF BYTE:=[16#4F,16#4B];
	arAnswerErr				: ARRAY[1..5] OF BYTE:=[16#45,16#52,16#52,16#4F,16#52];

	sDeleteSMS				: STRING(15);			(*Command-String*)
	arDeleteSMS				: ARRAY[1..15] OF BYTE; (*Command-ARRAY*)
	arDeleteSMSAnswerRcv	: ARRAY[1..200] OF BYTE;(*Received answer of the command*)
	arDeleteSMSAnswerClr	: ARRAY[1..200] OF BYTE;(*Empty-ARRAY to clear the answer for debugging*)
END_VAR


	rtrigStart(CLK:=bStart);

	tonTimeout();
	IF (tonTimeout.Q) THEN
		tonTimeout(IN := FALSE);
		nStep := 900;
	END_IF


	CASE nStep OF

	0: 	(*Idle Step*);
		tonTimeout(IN:=FALSE);
		IF (rtrigStart.Q AND NOT bBusy) THEN
			nStep := 5;
			bBusy := TRUE;
		ELSE
			bBusy := FALSE;
		END_IF


	5:
		bError					:= FALSE;
		nErrorId				:= 0;
		tonWaitTime				(IN := FALSE);
		tonTimeout				(IN := TRUE, PT := tTimeout);
		fbClearComBuffer		(buffer:=stRxBuffer);
		fbClearComBuffer		(buffer:=stTxBuffer);
		arDeleteSMSAnswerRcv	:= arDeleteSMSAnswerClr;

		nStep := 50;


	50:(*Create command-Arrays*)

		(*Delete-command*)
		sDeleteSMS:='AT+CMGD="';
		sDeleteSMS:=CONCAT(sDeleteSMS,USINT_TO_STRING(nIndex));
		sDeleteSMS:=CONCAT(sDeleteSMS,'"X');	(*The "X" is a placeholder in the send-string
												for the "CR" (Hex 0D) in the send-Array*)
		MEMCPY(ADR(arDeleteSMS),ADR(sDeleteSMS),LEN(sDeleteSMS)); (*Copy String to ARRAY*)
		arDeleteSMS[LEN(sDeleteSMS)]:=16#0D;	(*Place the "CR" in the array*)

		nStep	:= 100;


	100:(*Send delete-command*)
		fbSendData(
		pSendData:=ADR(arDeleteSMS),
		Length:= LEN(sDeleteSMS),
		TXbuffer:= stTxBuffer);

		IF NOT fbSendData.Busy THEN
			nStep:=110;
		END_IF

		IF  fbSendData.Error<>0 THEN
			bError:= TRUE;
			nErrorID:= fbSendData.Error;
			nStep:=1000;
		END_IF


	110:(*Wait for the answer*)
		fbReceiveData(
		pPrefix:= 0,
		LenPrefix:= 0,
		pReceiveData:= ADR(arDeleteSMSAnswerRcv),
		SizeReceiveData:= SIZEOF(arDeleteSMSAnswerRcv),
		Timeout:= t#1000ms,
		RXbuffer:= stRxBuffer);

		(*Telegram is received*)
		IF 			fbReceiveData.DataReceived
			AND NOT fbReceiveData.busy	THEN
						nStep:=120;
		END_IF


	120:(*Find an "OK" or an "ERROR"-Part in the answer*)
		uiAnalyzeAnswer	:=0;
		FOR i:= (SIZEOF(arDeleteSMSAnswerRcv)-5) TO 1 BY -1 DO
			IF 		arDeleteSMSAnswerRcv[i]		= arAnswerOK[1]
				AND arDeleteSMSAnswerRcv[i+1] 	= arAnswerOK[2]		THEN
					uiAnalyzeAnswer:=1;		(*Delete SMS successfully executed*)
				EXIT;

			ELSIF	arDeleteSMSAnswerRcv[i]		= arAnswerErr[1]
				AND arDeleteSMSAnswerRcv[i+1] 	= arAnswerErr[2]
				AND arDeleteSMSAnswerRcv[i+2] 	= arAnswerErr[3]
				AND arDeleteSMSAnswerRcv[i+3] 	= arAnswerErr[4]
				AND arDeleteSMSAnswerRcv[i+4] 	= arAnswerErr[5]	THEN
					uiAnalyzeAnswer:=2;		(*Delete SMS failed*)
				EXIT;
			END_IF
		END_FOR

		CASE uiAnalyzeAnswer OF
			0:(*Undefined Answer*)
				bError:= TRUE;
				nErrorID:= 16#8010;
				nStep:=1000;

			1:(*Delete SMS successfully executed*)
				nStep:=1000;

			2:(*Delete SMS failed*)
				bError:= TRUE;
				nErrorID:= 16#800F;
				nStep:=1000;
		END_CASE


	900:(*Timeout*)
		bError:= TRUE;
		nErrorID:= 16#8001;
		nStep:=1000;


	1000:(*Reset Receive-FB*)
		fbReceiveData(	Reset:=TRUE,RXbuffer:= stRxBuffer);
		tonWaitTime(IN:=TRUE, PT:=t#500ms);
		IF	tonWaitTime.Q	THEN
			fbReceiveData(	Reset:=FALSE,RXbuffer:= stRxBuffer);
			nStep:=1010;
		END_IF


	1010:(*Send/Receive successful -> Reset FBs*)
		fbClearComBuffer(buffer:=stRxBuffer);
		fbClearComBuffer(buffer:=stTxBuffer);
		nStep:=0;
		bBusy:=FALSE;

	END_CASE;

END_FUNCTION_BLOCK

// ---- 00_FunctionsBlocks/Communication/SMS/FB_DeleteAllSMS.TcPOU
FUNCTION_BLOCK FB_DeleteAllSMS
VAR_INPUT
	bStart					: BOOL;
END_VAR
VAR_OUTPUT
	bBusy					: BOOL;
	bError					: BOOL;
	nErrorID				: UINT;
END_VAR

VAR_IN_OUT
	stTxBuffer				: ComBuffer;
	stRxBuffer				: ComBuffer;
END_VAR

VAR
	rtrigStart				: R_TRIG;

	fbSendData				: SendData;
	fbReceiveData			: ReceiveData;
	fbClearComBuffer		: ClearComBuffer;

	i						: INT;
	uiAnalyzeAnswer			: UINT;
	nStep					: UINT; (* sequence state *)
	tonWaitTime				: TON;
	tonTimeOut				: TON;
	tTimeout				: TIME:=t#5s;

	arAnswerOK				: ARRAY[1..2] OF BYTE:=[16#4F,16#4B];
	arAnswerErr				: ARRAY[1..5] OF BYTE:=[16#45,16#52,16#52,16#4F,16#52];

	sDeleteSMS				: STRING(15);			(*Command-String*)
	arDeleteSMS				: ARRAY[1..15] OF BYTE; (*Command-ARRAY*)
	arDeleteSMSAnswerRcv	: ARRAY[1..200] OF BYTE;(*Received answer of the command*)
	arDeleteSMSAnswerClr	: ARRAY[1..200] OF BYTE;(*Empty-ARRAY to clear the answer for debugging*)
END_VAR


	rtrigStart(CLK:=bStart);

	tonTimeout();
	IF (tonTimeout.Q) THEN
		tonTimeout(IN := FALSE);
		nStep := 900;
	END_IF


	CASE nStep OF

	0: 	(*Idle Step*);
		tonTimeout(IN:=FALSE);
		IF (rtrigStart.Q AND NOT bBusy) THEN
			nStep := 5;
			bBusy := TRUE;
		ELSE
			bBusy := FALSE;
		END_IF


	5:
		bError					:= FALSE;
		nErrorId				:= 0;
		tonWaitTime				(IN := FALSE);
		tonTimeout				(IN := TRUE, PT := tTimeout);
		fbClearComBuffer		(buffer:=stRxBuffer);
		fbClearComBuffer		(buffer:=stTxBuffer);
		arDeleteSMSAnswerRcv	:= arDeleteSMSAnswerClr;

		nStep := 50;


	50:(*Create command-Arrays*)

		(*Delete-command*)
		sDeleteSMS:='AT+CMGD="';
		sDeleteSMS:=CONCAT(sDeleteSMS,'1,4');
		
		sDeleteSMS:=CONCAT(sDeleteSMS,'"X');	(*The "X" is a placeholder in the send-string
												for the "CR" (Hex 0D) in the send-Array*)
		MEMCPY(ADR(arDeleteSMS),ADR(sDeleteSMS),LEN(sDeleteSMS)); (*Copy String to ARRAY*)
		arDeleteSMS[LEN(sDeleteSMS)]:=16#0D;	(*Place the "CR" in the array*)

		nStep	:= 100;


	100:(*Send delete-command*)
		fbSendData(
		pSendData:=ADR(arDeleteSMS),
		Length:= LEN(sDeleteSMS),
		TXbuffer:= stTxBuffer);

		IF NOT fbSendData.Busy THEN
			nStep:=110;
		END_IF

		IF  fbSendData.Error<>0 THEN
			bError:= TRUE;
			nErrorID:= fbSendData.Error;
			nStep:=1000;
		END_IF


	110:(*Wait for the answer*)
		fbReceiveData(
		pPrefix:= 0,
		LenPrefix:= 0,
		pReceiveData:= ADR(arDeleteSMSAnswerRcv),
		SizeReceiveData:= SIZEOF(arDeleteSMSAnswerRcv),
		Timeout:= t#1000ms,
		RXbuffer:= stRxBuffer);

		(*Telegram is received*)
		IF 			fbReceiveData.DataReceived
			AND NOT fbReceiveData.busy	THEN
						nStep:=120;
		END_IF


	120:(*Find an "OK" or an "ERROR"-Part in the answer*)
		uiAnalyzeAnswer	:=0;
		FOR i:= (SIZEOF(arDeleteSMSAnswerRcv)-5) TO 1 BY -1 DO
			IF 		arDeleteSMSAnswerRcv[i]		= arAnswerOK[1]
				AND arDeleteSMSAnswerRcv[i+1] 	= arAnswerOK[2]		THEN
					uiAnalyzeAnswer:=1;		(*Delete SMS successfully executed*)
				EXIT;

			ELSIF	arDeleteSMSAnswerRcv[i]		= arAnswerErr[1]
				AND arDeleteSMSAnswerRcv[i+1] 	= arAnswerErr[2]
				AND arDeleteSMSAnswerRcv[i+2] 	= arAnswerErr[3]
				AND arDeleteSMSAnswerRcv[i+3] 	= arAnswerErr[4]
				AND arDeleteSMSAnswerRcv[i+4] 	= arAnswerErr[5]	THEN
					uiAnalyzeAnswer:=2;		(*Delete SMS failed*)
				EXIT;
			END_IF
		END_FOR

		CASE uiAnalyzeAnswer OF
			0:(*Undefined Answer*)
				bError:= TRUE;
				nErrorID:= 16#8010;
				nStep:=1000;

			1:(*Delete SMS successfully executed*)
				nStep:=1000;

			2:(*Delete SMS failed*)
				bError:= TRUE;
				nErrorID:= 16#800F;
				nStep:=1000;
		END_CASE


	900:(*Timeout*)
		bError:= TRUE;
		nErrorID:= 16#8001;
		nStep:=1000;


	1000:(*Reset Receive-FB*)
		fbReceiveData(	Reset:=TRUE,RXbuffer:= stRxBuffer);
		tonWaitTime(IN:=TRUE, PT:=t#500ms);
		IF	tonWaitTime.Q	THEN
			fbReceiveData(	Reset:=FALSE,RXbuffer:= stRxBuffer);
			nStep:=1010;
		END_IF


	1010:(*Send/Receive successful -> Reset FBs*)
		fbClearComBuffer(buffer:=stRxBuffer);
		fbClearComBuffer(buffer:=stTxBuffer);
		nStep:=0;
		bBusy:=FALSE;

	END_CASE;

END_FUNCTION_BLOCK

// ---- 00_FunctionsBlocks/Communication/SMS/FB_Login.TcPOU
FUNCTION_BLOCK FB_Login

VAR_INPUT
	bStart					: BOOL;
	
END_VAR
VAR_OUTPUT
	bBusy					: BOOL;
	bError					: BOOL;
	nErrorID				: UINT;
END_VAR

VAR_IN_OUT
	stTxBuffer				: ComBuffer;
	stRxBuffer				: ComBuffer;
END_VAR

VAR
	rtrigStart				: R_TRIG;

	fbSendData				: SendData;
	fbReceiveData			: ReceiveData;
	fbClearComBuffer		: ClearComBuffer;

	i						: UINT;
	nStep					: UINT; (* sequence state *)
	tonWaitTime				: TON;
	tonTimeOut				: TON;
	tTimeout				: TIME:=t#30s;

	arAnswerOK				: ARRAY[1..2] OF BYTE:=[16#4F,16#4B];
	arAnswerErr				: ARRAY[1..5] OF BYTE:=[16#45,16#52,16#52,16#4F,16#52];

	sEchoOff				: STRING(5);			(*Command-String*)
	arEchoOff				: ARRAY[1..5] OF BYTE;	(*Command-ARRAY*)
	arEchoOffAnswerRcv		: ARRAY[1..5] OF BYTE;	(*Received answer of the command*)
	arEchoOffAnswerClr		: ARRAY[1..5] OF BYTE;	(*Empty-ARRAY to clear the answer for debugging*)

	sLogin					: STRING(21);			(*Command-String*)
	arLogin					: ARRAY[1..21] OF BYTE;	(*Command-ARRAY*)
	arLoginAnswerRcv		: ARRAY[1..5] OF BYTE;	(*Received answer of the command*)
	arLoginAnswerClr		: ARRAY[1..5] OF BYTE;	(*Empty-ARRAY to clear the answer for debugging*)
END_VAR

	rtrigStart(CLK:=bStart);  //Rising Edge detect

	tonTimeout();
	IF (tonTimeout.Q) THEN
		tonTimeout(IN := FALSE);
		nStep := 900;
	END_IF


	CASE nStep OF

	0: 	(*Idle Step*);
		tonTimeout(IN:=FALSE);
		tonWaitTime(IN:=FALSE);
		IF (rtrigStart.Q AND NOT bBusy) THEN
			nStep := 5;
			bBusy := TRUE;
		ELSE
			bBusy := FALSE;
		END_IF


	5:
		bError				:= FALSE;
		nErrorId			:= 0;
		tonTimeout			(IN := TRUE, PT := tTimeout);
		fbClearComBuffer	(buffer:=stRxBuffer);
		fbClearComBuffer	(buffer:=stTxBuffer);
		arEchoOffAnswerRcv	:= arEchoOffAnswerClr;
		arLoginAnswerRcv	:= arLoginAnswerClr;
	//	MEMSET(ADR(sMessageText),0,SIZEOF(sMessageText));
		nStep := 50;


	(*10:(*Length PIN-number within range?*)
		IF 		LEN(sPinNumber) < 1
			OR	LEN(sPinNumber) > 10 THEN
			bError		:= TRUE;
			nErrorID	:= 16#8002;
			nStep		:= 1000;
		ELSE
			nStep		:= 20;
		END_IF


	20:(*Phone-number contains correct characters? 0..9*)
		FOR i:=1 TO LEN(sPinNumber) DO
			IF 		ASC(MID(sPinNumber,1,i)) < 16#30
				OR	ASC(MID(sPinNumber,1,i)) > 16#39	(*a non-numeric character in PIN*)	THEN
				bError		:= TRUE;
				nErrorID	:= 16#8003;
			END_IF
		END_FOR

		IF bError	THEN
			nStep	:= 1000;
		ELSE
			nStep	:= 50;
		END_IF*)


	50:(*Create command-Arrays*)

		(*Echo OFF*)
		sEchoOff:='ATE0';
		sEchoOff:=CONCAT(sEchoOff,'X');	(*The "X" is a placeholder in the send-string
										for the "CR" (Hex 0D) in the send-Array*)
		MEMCPY(ADR(arEchoOff),ADR(sEchoOff),LEN(sEchoOff)); (*Copy String to ARRAY*)
		arEchoOff[LEN(sEchoOff)]:=16#0D;(*Place the "CR" in the array*)

		(*Mode Text*)
		sLogin:='AT+CMGF=';
		sLogin:=CONCAT(sLogin,'1');
		sLogin:=CONCAT(sLogin,'X');	(*The "X" is a placeholder in the send-string
										for the "CR" (Hex 0D) in the send-Array*)
		MEMCPY(ADR(arLogin),ADR(sLogin),LEN(sLogin)); (*Copy String to ARRAY*)
		arLogin[LEN(sLogin)]:=16#0D;	(*Place the "CR" in the array*)

		nStep	:= 100;


	100:(*Turn Off the Echo*)
		fbSendData(
		pSendData:=ADR(arEchoOff),
		Length:= LEN(sEchoOff),
		TXbuffer:= stTxBuffer);

		IF NOT fbSendData.Busy THEN
			nStep:=110;
		END_IF

		IF  fbSendData.Error<>0 THEN
			bError:= TRUE;
			nErrorID:= fbSendData.Error;
			nStep:=1000;
		END_IF


	110:(*Wait explicitly (by Prefix) for an "OK"-Answer,
		because the echo may still be on or is already switched off, so the answer may differ in length.
		Only ok is possible, any other answer caused by Comm-Error will end in global timeout*)

		fbReceiveData(
		pPrefix:= ADR(arAnswerOK),
		LenPrefix:= 2,
		pReceiveData:= ADR(arEchoOffAnswerRcv),
		SizeReceiveData:= SIZEOF(arEchoOffAnswerRcv),
		Timeout:= t#500ms,
		RXbuffer:= stRxBuffer);

		(*Telegram is received*)
		IF 			fbReceiveData.DataReceived
			AND NOT fbReceiveData.busy
			AND		(arEchoOffAnswerRcv[1]=arAnswerOK[1])
			AND 	(arEchoOffAnswerRcv[2]=arAnswerOK[2])	THEN
						nStep:=200;
		END_IF


	200:(*Send AT+CMGF Command*)
		fbSendData(
		pSendData:=ADR(arLogin),
		Length:= LEN(sLogin),
		TXbuffer:= stTxBuffer);

		IF NOT fbSendData.Busy THEN
			nStep:=210;
		END_IF

		IF  fbSendData.Error<>0 THEN
			bError:= TRUE;
			nErrorID:= fbSendData.Error;
			nStep:=1000;
		END_IF


	210:(*Wait for OK or Err-Answer. Any other answer caused by Comm-Error will end in global timeout*)
		(*Do NOT remove the "0" prefix, because the FB is used previously*)
		fbReceiveData(
		pPrefix:= 0,
		LenPrefix:= 0,
		pReceiveData:= ADR(arLoginAnswerRcv),
		SizeReceiveData:= SIZEOF(arLoginAnswerRcv),
		Timeout:= t#500ms,
		RXbuffer:= stRxBuffer);

		(*Telegram is received*)
		IF 	(fbReceiveData.DataReceived	AND NOT 	fbReceiveData.busy)	THEN
				nStep:=220;
		END_IF


	220:(*Analyze answer*)
		IF		(arLoginAnswerRcv[3]=arAnswerOK[1]) AND (arLoginAnswerRcv[4]=arAnswerOK[2])	THEN
					nStep:=1000;		(*Login successful*)
		ELSIF	(arLoginAnswerRcv[3]=arAnswerErr[1]) AND (arLoginAnswerRcv[4]=arAnswerErr[2])	THEN
					bError:= TRUE;
					nErrorID:= 16#8004;	(*Login failed due to wrong PIN or no Card or already logged in*)
					nStep:=1000;
		ELSE
					bError:= TRUE;
					nErrorID:= 16#8005;	(*Undefined answer*)
					nStep:=1000;
		END_IF


	900:(*Timeout*)
		bError:= TRUE;
		nErrorID:= 16#8001;
		nStep:=1000;


	1000:(*Reset Receive-FB*)
		fbReceiveData(	Reset:=TRUE,RXbuffer:= stRxBuffer);
		tonWaitTime(IN:=TRUE, PT:=t#1000ms);
		IF	tonWaitTime.Q	THEN
			tonWaitTime(IN:=FALSE);
			fbReceiveData(	Reset:=FALSE,RXbuffer:= stRxBuffer);
			nStep:=1010;
		END_IF


	1010:(*Send/Receive successful -> Reset FBs*)
		fbClearComBuffer(buffer:=stRxBuffer);
		fbClearComBuffer(buffer:=stTxBuffer);
		tonWaitTime(IN:=TRUE, PT:=t#1000ms);
		IF	tonWaitTime.Q	THEN
			tonWaitTime(IN:=FALSE);
			nStep:=0;
			bBusy:=FALSE;
		END_IF

	END_CASE;

END_FUNCTION_BLOCK

// ---- 00_FunctionsBlocks/DataProcessing/FB_XorWord.TcPOU
FUNCTION_BLOCK FB_XorWord
// Takes in a Word and its past value and input the bits that have changed and the bits active in 2 arrays of array of bool
VAR_INPUT
	MyNewWord	:WORD;      //Mon nouveau AlarmCode actualisée a chaque temps de Cycle
	MyWord		:WORD;		// AlarmCode du cycle précedent
END_VAR
VAR_OUTPUT
	XORarray 	:ARRAY [0..15] OF BOOL;  //Tableau avec les bits qui ont subit une modif entre MyNewWord et MyWord
	Boolarray	:ARRAY [0..15] OF BOOL; // MyNewWord convertis en Array of BOOL
END_VAR
VAR
	MyXorWord:WORD;
	FB_Word_TO_Bool : FB_WordToArrayOfBool;
END_VAR

// Operateur XOR pour trouver les Bits modifiés
MyXorWord:= Myword XOR MyNewWord;

FB_Word_TO_Bool(MyWord:=MyXorWord,ArrayOfBool=>XORarray);
FB_Word_TO_Bool(MyWord:=MyNewWord,ArrayOfBool=>Boolarray);

END_FUNCTION_BLOCK

// ---- 00_FunctionsBlocks/BoolManagement/FB_WordToArrayOfBool.TcPOU
FUNCTION_BLOCK FB_WordToArrayOfBool
// Transforms a Word in an array of BOOL;
VAR_INPUT
	MyWord	:WORD;
END_VAR
VAR_OUTPUT
	ArrayOfBool: ARRAY [0..15] OF BOOL;
END_VAR

ArrayOfBool[0] := BIT_TO_BOOL(MyWord.0);
ArrayOfBool[1] := BIT_TO_BOOL(MyWord.1);
ArrayOfBool[2] := BIT_TO_BOOL(MyWord.2);
ArrayOfBool[3] := BIT_TO_BOOL(MyWord.3);
ArrayOfBool[4] := BIT_TO_BOOL(MyWord.4);
ArrayOfBool[5] := BIT_TO_BOOL(MyWord.5);
ArrayOfBool[6] := BIT_TO_BOOL(MyWord.6);
ArrayOfBool[7] := BIT_TO_BOOL(MyWord.7);
ArrayOfBool[8] := BIT_TO_BOOL(MyWord.8);
ArrayOfBool[9] := BIT_TO_BOOL(MyWord.9);
ArrayOfBool[10] := BIT_TO_BOOL(MyWord.10);
ArrayOfBool[11] := BIT_TO_BOOL(MyWord.11);
ArrayOfBool[12] := BIT_TO_BOOL(MyWord.12);
ArrayOfBool[13] := BIT_TO_BOOL(MyWord.13);
ArrayOfBool[14] := BIT_TO_BOOL(MyWord.14);
ArrayOfBool[15] := BIT_TO_BOOL(MyWord.15);

END_FUNCTION_BLOCK

// ---- 00_FunctionsBlocks/Communication/SMS/FB_Extract_Num_Mes.TcPOU
FUNCTION_BLOCK FB_Extract_Num_Mes
// extract phone number from the received message
VAR_INPUT
    InMessage     : STRING(255);
END_VAR
VAR_OUTPUT
    OutDataEntry  :ST_SMSDataSetEntry_Read;
END_VAR
VAR
    ChaineTmp     : STRING(255);
    Num           : STRING(255);
    Pos           : INT;
    Pos1          : INT;
    Pos2          : INT;
    Pos3          : INT;    
	Offset		: INT ; 
END_VAR

//+CMGR: "REC UNREAD","+33776039883",,"18/04/19,18:25:44+08"$R$NBonjour je m'appelle henry$R$N 50
Pos:=FIND(InMessage,',"');
chaineTmp:=MID(InMessage,LEN(InMessage)-21,POS+2);
Pos1:=FIND(chaineTmp,'",,');
Num:=MID(chaineTmp,Pos1-1,1);
Pos3:= FIND(Num,'+');
OutDataEntry.Num:= SEL(Pos3= 0 ,Num ,CONCAT(STR1:= CstPhoneIndicator_G, STR2:= Num) );
Pos2:=FIND(InMessage,'$R$N');
Offset := FIND(MID(InMessage,LEN(InMessage)-Pos2,Pos2+2),'$R$N') ;


OutDataEntry.Message:=MID(InMessage,Offset-1,Pos2+2);//OutDataEntry.Message:=MID(InMessage,LEN(InMessage)-Pos2-3,LEN(InMessage));	// OutDataEntry.Message:=MID(InMessage,LEN(InMessage)-Pos2-3,Pso2+2);

END_FUNCTION_BLOCK

// ---- 00_FunctionsBlocks/Annexesfunction/FUN_ConnectVPN.TcPOU
PROGRAM FUN_ConnectVPN

VAR_INPUT
	ParamNetID				: STRING :='' ; // Unit ID of the PC with internet connexion
	IN_CmdStart 			: BOOL;
	IN_DirExe				: STRING;
	IN_OpenVpnFile			: STRING;
END_VAR
VAR_OUTPUT
	OUT_Completed			: BOOL;
END_VAR

VAR
	RS_Start				: RS;
	TRIG_Completed			: R_TRIG;
	TRIG_Start				: R_TRIG;
	start_process			: NT_StartProcess;
	TRIG_Available			: F_TRIG;
	bTest: BOOL;
END_VAR


TRIG_Start(CLK := IN_CmdStart);

start_process
(
	NETID := ParamNetID,
	PATHSTR := '"C:\Program Files\OpenVPN\bin\openvpn-gui.exe"',
	DIRNAME := 'C:\Program Files\OpenVPN\bin',
	COMNDLINE := Concat(str1 := '--command connect ', str2 := concat(STR1 := IN_OpenVpnFile, STR2 := '.ovpn')),
	Start := TRIG_Start.Q
);

END_PROGRAM

// ---- 00_FunctionsBlocks/Annexesfunction/FUN_DisconnectVPN.TcPOU
PROGRAM FUN_DisconnectVPN

VAR_INPUT
	ParamNetID				: STRING :='' ; // Unit ID of the PC with internet connexion
	IN_CmdStart 			: BOOL;
	IN_DirExe				: STRING;
END_VAR
VAR_OUTPUT
	OUT_Completed			: BOOL;
END_VAR

VAR
	TRIG_Start				: R_TRIG;
	start_process			: NT_StartProcess;
END_VAR

TRIG_Start(ClK := IN_CmdStart);

start_process
(
	NETID := ParamNetID,
	PATHSTR := '"c:\Program Files\OpenVPN\bin\openvpn-gui.exe" ',
	DIRNAME := 'C:\Program Files\OpenVPN\bin',
	COMNDLINE := '--command disconnect_all',
	Start := TRIG_Start.Q
);

END_PROGRAM

// ---- 00_FunctionsBlocks/Annexesfunction/FUN_GetPublicIp.TcPOU
PROGRAM FUN_GetPublicIp

VAR_INPUT
	ParamNetID				: STRING :='' ; // Unit ID of the PC with internet connexion
	IN_CmdStart 			: BOOL;
	IN_DirExe				: STRING;
END_VAR
VAR_OUTPUT
	OUT_Completed			: BOOL;
END_VAR

VAR
	RS_Start				: RS;
	TRIG_Completed			: R_TRIG;
	TRIG_Start				: R_TRIG;
	start_process			: NT_StartProcess;
END_VAR


TRIG_Start(ClK := IN_CmdStart);
TRIG_Completed(CLK := OUT_Completed);


RS_Start(SET := TRIG_Start.Q, RESET1 := TRIG_Completed.Q);

IF RS_Start.Q1 THEN
	IN_CmdStart := FALSE;
	start_process
	(
		NETID := ParamNetID,
		PATHSTR := Concat(IN_DirExe, 'GetPublicIp.exe'),
		DIRNAME := IN_DirExe,
		COMNDLINE := '',
		Start := TRUE
	);
ELSE
	start_process(START := FALSE);
END_IF

IF TRIG_Completed.Q THEN
	OUT_Completed := FALSE;
END_IF

END_PROGRAM

// ---- 00_FunctionsBlocks/Annexesfunction/FUN_PingHost.TcPOU
PROGRAM FUN_PingHost
VAR_INPUT
	IN_bStart			: BOOL;	
	IN_PingAdr			: STRING(50);
	IN_DirBatLocation	: STRING(255);
END_VAR
VAR_OUTPUT
	OUT_Result			: BOOL;
	OUT_Completed 		: BOOL;
	OUT_Busy			: BOOL;
	OUT_Error			: BOOL;
END_VAR
VAR
	ReadLine			: T_MaxString;
	ReadResult 			: T_MAXString;
	StartProcess 		: NT_StartProcess;
	TP_StartFunction	: TP;
	TP_StartProcess		: TP;
	RS_Start			: RS;
	Trig_Start			: R_TRIG;
	FB_Read 			: FB_READ;
	Outvalue			: STRING(255);
END_VAR

Trig_Start(CLK := IN_bStart);
IF Trig_Start.Q THEN 
	ReadResult := '';
END_IF
RS_Start(Set := Trig_Start.Q, RESET1 := OUT_Completed);
OUT_Busy := FALSE;
OUT_Completed := FALSE;

IF RS_Start.Q1 THEN
	//Phase de start du processus
	OUT_Busy := TRUE;
	TP_StartProcess(IN := RS_Start.Q1, PT := T#7S);
	StartProcess
	(
		NETID := '',
		PATHSTR:= CONCAT(IN_DirBatLocation, 'PingHost.bat'),
		DIRNAME := IN_DirBatLocation,
		COMNDLINE := IN_PingAdr,
		Start := RS_Start.Q1,
		TMOUT := T#7S
	);
	
	//Phase d'analyse du processus
	IF NOT StartProcess.BUSY AND NOT StartProcess.ERR  AND NOT TP_StartProcess.Q THEN
		FB_Read
		(
			InDirectory := CONCAT(IN_DirBatLocation, 'Ping.txt'),
			InExecute := TRUE,
			OutValue => ReadLine
		);
		
		IF NOT FB_Read.OutbBusy AND NOT fb_read.OutError THEN
			OUT_Completed := TRUE;
			OUT_Busy := FALSE;
			TP_StartProcess(in := FALSE);
			FB_Read(InExecute := FALSE);
			StartProcess(Start := FALSE);
			
			IF left(ReadLine, 14) = 'host reachable' THEN
				ReadResult := 'PING OK';
				OUT_Result := TRUE;
			ELSE
				OUT_Result := FALSE;
				ReadResult := 'PING NOT OK';

			END_IF
		END_IF
	ELSIF NOT StartProcess.BUSY AND StartProcess.ERR THEN
		Out_Error := TRUE;
	END_IF
END_IF

END_PROGRAM

// ---- 00_FunctionsBlocks/DataProcessing/ReadFile/FB_Read.TcPOU
FUNCTION_BLOCK FB_Read
//Permet de lire les Valeurs de max 1 semaine de points (1 pt/min pdt 7 jours)

VAR_INPUT
	InDirectory 				: T_MaxString;		// Base file of the Historization 
	InExecute					: BOOL;			//Rising Edge detection of read
END_VAR                 		

VAR_OUTPUT              		
	OutValue					: T_MaxString;
	OutCompleted				: BOOL;
	OutbBusy					: BOOL;
	OutError 					: BOOL;
	OutErrorID 					: UINT; // 1 : File not found

END_VAR                 		
VAR     
	// Initialisation 
	RS_Busy						: RS;
	Trig_Start 					: R_TRIG;
	FullDirectory				: STRING;  
	
	OpenFile					: FB_FileOpen;
	ReadFile					: FB_FileRead;
	CloseFile					: FB_FileClose;
	
	Opening						: BOOL := TRUE;
	Reading						: BOOL;
	Closing						: BOOL;
	
	EOF_Reached					: BOOL;
	
	FileHandle					: UINT;
	FileHandle_Old				: UINT;
	
	NbJours						: UINT;
	KK: UINT 					:= 1;
END_VAR

Trig_Start(CLK := InExecute);

IF Trig_Start.Q THEN 
	Outerror:= FALSE ; // On reinitialize l'error à un nouvel essai . 
	OpenFile(bExecute:= FALSE  ); 
END_IF

RS_Busy(Set := Trig_Start.Q, RESET1 := Outerror OR OutCompleted);
OutbBusy := RS_Busy.Q1;
OutCompleted := FALSE;


IF RS_Busy.Q1 THEN	
		//Ouverture du Fichier, récupération du handle
		OpenFile
		(
			sNetId := '',
			sPathName := InDirectory,
			nMode := FOPEN_MODEREAD,
			ePath := PATH_GENERIC,
			bExecute := TRUE,
			hFile => FileHandle
		);
		
		IF NOT OpenFile.bBusy AND OpenFile.bError AND OpenFile.nErrId = 1804 THEN // Le fichier n'existe pas 
			OutErrorID := 1;
			OutError := OpenFile.bError;
		ELSIF OpenFile.bError THEN		// Il y a eu une autre erreur
			OutError := OpenFile.bError;
		ELSIF NOT OpenFile.bError AND NOT OpenFile.bBusy AND FileHandle <> 0 THEN
			opening := FALSE;
		END_IF
		
		
		
		IF NOT opening AND NOT EOF_Reached THEN			
			ReadFile
			(
				sNetId := '',
				hFile := FileHandle,
				bExecute := TRUE,
				tTimeout := T#1S,
				pReadBuff := ADR(OutValue),
				cbReadLen := SIZEOF(OutValue),				
				bEOF => EOF_Reached
			);	
			IF NOT ReadFile.bBusy AND ReadFile.bError THEN
				OutError := TRUE;	
				ReadFile(bExecute := FALSE);
			ELSIF NOT ReadFile.bBusy THEN
				ReadFile(bExecute := FALSE);	
			END_IF
		ELSIF EOF_Reached THEN
			ReadFile(bExecute := FALSE);
	
			CloseFile
			(
				sNetId := '',
				bExecute := TRUE,
				hFile := FileHandle,
				tTimeout := T#1S
			);
			IF NOT CloseFile.bBusy AND NOT CloseFile.bError  THEN
				Opening := TRUE;
				EOF_Reached := FALSE;
				OpenFile(bExecute := FALSE);
				ReadFile(bExecute := FALSE);
				CloseFile(bExecute := FALSE);
				
				OUTCompleted := TRUE;
			ELSIF CloseFile.bError THEN
				OutError := TRUE;
				OutErrorID := UDINT_TO_UINT(Closefile.nErrId);
			END_IF	
		END_IF
	END_IF

END_FUNCTION_BLOCK

// ---- 00_FunctionsBlocks/Annexesfunction/PRG_RestartPlc.TcPOU
PROGRAM PRG_RestartPlc
VAR
END_VAR
VAR_INPUT
	CmdRestart 	: BOOL;
END_VAR

VAR
	RestartProcess : NT_Reboot;
	Trig_Restart	: R_TRIG;
	
END_VAR

Trig_Restart(CLK := CmdRestart);

RestartProcess
(
	NETID := '',
	START := Trig_Restart.Q,
	DELAY := 5,
	TMOUT := T#1S
);

END_PROGRAM

// ---- 00_FunctionsBlocks/Annexesfunction/PRG_RestartService.TcPOU
PROGRAM PRG_RestartService
// FB to Compress all files of the directory. 
VAR_INPUT
	IN_Directory			: T_MaxString; // directory of the file to compress
	ParamNetID				: STRING ; // Net ID of the PC with HH collector
	IN_ServiceName			: STRING  ;
	Start					: BOOL;
END_VAR
VAR
	StartProcess 			: NT_StartProcess;
	TrigStart				: R_TRIG;
END_VAR

TrigStart(CLK:=Start);
	StartProcess
	(
		NETID := ParamNetID,
		PATHSTR := concat(str1:= IN_Directory, str2 := 'IN_ServiceName'),
		DIRNAME := IN_Directory,
		COMNDLINE := '',
		Start := TrigStart.Q,
		TMOUT := T#3M
	);
	IF NOT StartProcess.BUSY THEN
		IF NOT StartProcess.ERR THEN
			StartProcess(Start := FALSE);
		ELSE
			StartProcess(Start := FALSE);
		END_IF
	END_IF

END_PROGRAM

// ---- 00_FunctionsBlocks/BoolManagement/FB_CountNinTimeWindow.TcPOU
FUNCTION_BLOCK FB_CountNinTimeWindow
VAR_INPUT
	IN_CountMax			: UINT := 3 ; 
	IN_bInput				: BOOL;
	IN_bReset			: BOOL;
END_VAR
VAR_OUTPUT
	OUT_FlagNinT		: BOOL;		// Output : if CountMax Input occured in the last T min, this variable = TRUE;
END_VAR
VAR
	TimeFault1			: TIME;		// Temps du troisième défaut GTE (chronologiquement parlant)
	TimeFault2			: TIME;		// Temps du deuxième défaut GTE (chronologiquement parlant)
	TimeFault3			: TIME;		// Temps du premier défaut GTE (chronologiquement parlant)
	TriggerGTE			: R_TRIG;	
	
	TestDiff			: TIME;
END_VAR
VAR_INPUT PERSISTENT
	ParamTimeToMeasure	: TIME := T#30M; // Time during which the 3 GTE are measured. Used for testing.
END_VAR

TriggerGTE(CLK:= IN_bInput);

 IF IN_bReset THEN
		OUT_FlagNinT := FALSE;
		TimeFault1 := T#0S;
		TimeFault2 := T#0S;
		TimeFault3 := T#0S;
END_IF

IF TriggerGTE.Q AND TimeFault3 = T#0S THEN
	TimeFault3 := TIME();
ELSIF TriggerGTE.Q AND TimeFault2 = T#0S THEN
	TimeFault2 := TIME();
ELSIF TriggerGTE.Q AND TimeFault1 = T#0S THEN
	TimeFault1 := TIME();
ELSIF TriggerGTE.Q THEN
	TimeFault3 := TimeFault2;
	TimeFault2 := TimeFault1;
	TImeFault1 := TIME();
END_IF


IF TimeFault1 - TimeFault3 < ParamTimeToMeasure AND TimeFault1 <> T#0S THEN
	OUT_FlagNinT := TRUE;
ELSE 
	OUT_FlagNinT := FALSE;
END_IF

END_FUNCTION_BLOCK

// ---- 00_FunctionsBlocks/BoolManagement/FB_TapVariable.TcPOU
FUNCTION_BLOCK FB_TapVariable
////////////////// 
// TAp a variable when input is active and reset after 
//////////////////	

VAR_IN_OUT
	TapOut			: BOOL;		// Output VTap Variable
	
END_VAR

VAR_INPUT
	TapTrigger		: BOOL;		// Input Trigger
	
END_VAR

VAR
	F_TRIG_Trigger	: F_TRIG;	// Trigger detection 
	R_TRIG_Trigger	: R_TRIG;	// Trigger detection 		
	
	
END_VAR

R_TRIG_Trigger(CLK:= TapTrigger);
F_TRIG_Trigger(CLK:= TapTrigger);

IF R_TRIG_Trigger.Q THEN
	TapOut			:=TRUE;
	
ELSIF F_TRIG_Trigger.Q  THEN 
	TapOut			:=FALSE ;
			
END_IF

END_FUNCTION_BLOCK

// ---- 00_FunctionsBlocks/BoolManagement/FB_Toggle2Tap.TcPOU
FUNCTION_BLOCK FB_Toggle2Tap
///////////
// FB to change a toggle into a tap with constant duration//
///////////

VAR_INPUT
	TapDuration		: TIME; 	// (s) Tap duration
	
	ToggleVar 		: BOOL;		// Toggled input variable 

	
END_VAR

VAR_OUTPUT
	TapVar			: BOOL ; 	// Tapped output variable
	
END_VAR

VAR				
	R_TRIG			: R_TRIG ;				// Create a square at Rising Edge Detection
	F_TRIG			: F_TRIG ;				// Create a square at falling Edge Detection 
	TP				: TP ; 					// Square Signal 

END_VAR

R_TRIG(CLK := ToggleVar) ;  							// Rising Edge Detection
F_TRIG(CLK := ToggleVar) ; 								// Falling Edge Detection

TP(IN := R_TRIG.Q OR F_TRIG.Q , PT := TapDuration) ;  	// Square signal 

TapVar		:= TP.Q ; 									// OUtput variable

END_FUNCTION_BLOCK

// ---- 00_FunctionsBlocks/BoolManagement/FB_WriteOnChange.TcPOU
FUNCTION_BLOCK FB_WriteOnChange
////////////////// 
// Write output variable , equals to input variable only if input variable changed state 
//////////////////	

VAR_INPUT
	Size			: UDINT; 				// Variable size 
	VarOut			: POINTER TO BYTE;		// Output  Variable Memory Address
	VarInput		: POINTER TO BYTE;		// Input Variable Memory Address	
END_VAR


VAR
	VarHold 		: DWORD  ; 	

END_VAR

IF MEMCMP(pBuf1:= VarInput, pBuf2:= ADR(VarHold) , n:=Size )<>0  THEN
	MEMCPY(srcAddr:= VarInput , destAddr := VarOut, n:= Size ) ;
END_IF

IF MEMCMP(pBuf1:= VarOut, pBuf2:= ADR(VarHold) , n:=Size )<>0  THEN
	MEMCPY(srcAddr:= VarOut , destAddr := VarInput, n:= Size ) ;
END_IF

MEMCPY(srcAddr:= VarInput , destAddr := ADR(VarHold), n:= Size ) ;

END_FUNCTION_BLOCK

// ---- 00_FunctionsBlocks/BoolManagement/RS_NoReset.TcPOU
FUNCTION_BLOCK RS_NoReset
//Output reset the input if the input is false 
VAR_INPUT
	Set 		: BOOL;
	Reset 		: BOOL;
END_VAR
VAR_OUTPUT
	Q1 			: BOOL;
END_VAR
VAR
	TRIG 		: R_TRIG;
	RS 			: RS;
END_VAR

TRIG(CLK := Set);
RS(Set := TRIG.Q, RESET1 := Reset AND NOT Set, Q1 => Q1);

END_FUNCTION_BLOCK

// ---- 00_FunctionsBlocks/Communication/IEC104/FB_IEC104ServerAkuo.TcPOU
FUNCTION_BLOCK FB_IEC104ServerAkuo
VAR_INPUT
	protPara  		: ST_IEC870_5_104ProtocolParams ;	// protocol parameters 
	sysPara	  		: ST_IEC870_5_101SystemParams ; 	// system parameters. 
	akuoPara		: ST_IEC104AkuoParam;				// akuo parameters. 
	
	IN_bEnable		: BOOL := TRUE ;					// enable or disable IEC 104 Server  .
	IN_Local		: BOOL ;  							// Server in local. Data flow is inhibated in control direction, allow in monitor direction.  
	IN_CmdReset		: BOOL ;							// Reset after a change in the protPara , or  sysPara
	
	memory 			: PVOID ; 							// ADR() . Pointer to starting address. 	
	AODB 			: ARRAY[0..GVL_Cst.CstNbAOEntries] OF ST_IEC870_5_101AODBEntry ;	// AODB	
END_VAR

VAR_OUTPUT
	eConnState		: E_SocketConnectionState := eSOCKET_DISCONNECTED;
	eDTState		: E_IEC870_5_104DataTransferState := eIEC870_STOPDT ;
END_VAR
VAR
// M_INIT 
	bInit					: BOOL := TRUE;

//M_PREPAREAO // 
	nBytesRead				: ARRAY[0..GVL_Cst.CstNbAOEntries] OF UDINT;		// Number of bytes taken by the raw data ( float = 4  SIQ = 1 , ...)
	Mask					: ARRAY[0..GVL_Cst.CstNbAOEntries] OF  DWORD;		// Mask corresponding to number of byte above . 
	MesCmd_old				: ARRAY[0..GVL_Cst.CstNbAOEntries] OF DWORD ; 		// Value in the memory space ( after bytes and bit offset ). 
	MesDword_Old			: ARRAY[0..GVL_Cst.CstNbAOEntries] OF DWORD;		// Raw dword value in memory space . 
	FB_Flicker				: ARRAY[0..GVL_Cst.CstNbAOEntries] OF FB_DetectFlicker ; 	// Function to detect flickering 

// M_CONNECT //
	hServer					: T_HSERVER; // TCP/IP server handle
	eComState				: E_ComState	:= INIT;
	fbConnection			: FB_ServerClientConnection;
	fbProtocol				: FB_IEC870_5_104TProtocol;

// TIME MANAGEMEMENT //
	systemTime_CP56Time2a			: T_CP56Time2a;
	FB_LocalSystTime				: FB_LocalSystemTime;
	CalLocalTimeStruct				: TIMESTRUCT ; 
	
// PROCESS DATA 
	stBuffer				: ST_IEC870_5_101TBuffer;		// Buffer of data to send in monitoring direction
	fbBuffer				: FB_IEC870_5_101TBufferCtrl;	// Buffer of data to send in control direction . 
	
	stTxAsdu 				: ST_IEC870_5_101AOGen; 	// asdu to be send . Copied from current AO . 
	KK						: INT ;	// loop 
	JJ						: INT;	// loop
	
// M_READCMD //
	stRxAsdu 				: ST_IEC870_5_101AOGen; // received asdu 
	nQOI					: BYTE;		// general interrogation data
	fbsetLocalTime			: NT_SetLocalTime; //clock synchronisation time apply

// M_CYCLIC // 
	fbCyclicTime				: TON;	// Cyclic trigger

//M_CHANGE DATA//
	CmdOldValue				: ARRAY[0..GVL_Cst.CstNbAOEntries] OF DWORD;		// Value of predecessing commAND  

END_VAR

IF bInit OR IN_CmdReset THEN 
	M_Init() ;
	bInit := FALSE ; 
END_IF

M_PrepareAO(); 

// GET LOCAL TIME AND CONVERT TO CP56Time 
FB_LocalSystTime(
	bEnable := TRUE,
	dwCycle := 1,
	systemTime => CalLocalTimeStruct);
		 
systemTime_CP56Time2a := SYSTEMTIME_TO_CP56Time2a(TIMESTR := CalLocalTimeStruct, SU := FALSE);

// Connexion management 
M_Connect();

// Read Command in control direction//
M_ReadCmd() ;

// Cyclic Data in monitoring direction//
fbCyclicTime(IN:= sysPara.bPerCyclic XOR fbCyclicTime.Q, PT:= sysPara.tPerCyclicBase);
IF sysPara.bPerCyclic AND fbCyclicTime.Q AND (eComState = DATATRANSFER) THEN
	M_Cyclic();
END_IF

// On change data in monitoring direction//
IF (eComState = DATATRANSFER) THEN
	M_ChangeData();
END_IF

METHOD M_ChangeData : BOOL
VAR_INPUT
END_VAR
FOR KK := 0 TO akuoPara.iAOnb DO 
	IF AODB[KK].aObj.obj.ident.eType = 30 OR AODB[KK].aObj.obj.ident.eType = 31 THEN 
		// Get value of corresponding byte .
		IF CmdOldValue[KK]<> MesCmd_old[KK] THEN 
			CmdOldValue[KK] := MesCmd_old[KK] ;
			stTxAsdu :=  AODB[KK].aObj.obj ; 
			stTxAsdu.ident.eCOT		:= eIEC870_COT_SPONTAN;	// cause of transmission - spontaneous
			stTxAsdu.ident.nORG		:= sysPara.orgAddr;				// originator address

			fbBuffer.TxAddObj(putObj := stTxAsdu,buffer := stBuffer);
			IF NOT fbBuffer.bOk THEN
				// code for buffer overflow
				RETURN; 
			END_IF	 		
		END_IF
	END_IF
END_FOR
END_METHOD

METHOD M_Connect : BOOL
VAR_INPUT
END_VAR

VAR

END_VAR
// connection management
CASE eComState OF
INIT: 
	// INIT protocol parameter
	fbConnection.eMode		:= eACCEPT_ALL;	// accept all incomming connections
	fbConnection.tReconnect	:= T#2S;
	
	fbProtocol.sSrvNetID				:= '';		
	fbProtocol.protPara.bPackFrames		:= TRUE;
	fbProtocol.protPara.bThrottleMode	:= protPara.bThrottleMode;
	fbProtocol.bOutDbg					:= FALSE;	// disable debug output


	// INIT RX/TX buffer parameter
	stBuffer.eDbg					:= eIEC870_FIFO_DBG_ALL;
	stBuffer.asduFmt.eCOTSize		:= eIEC870_COT_TwoOctets;		// cause of transfer size
	stBuffer.asduFmt.eAsduAddrSize	:= eIEC870_AsduAddr_TwoOctets;	// common asdu addr size
	stBuffer.asduFmt.eObjAddrSize	:= eIEc870_ObjAddr_ThreeOctets;	// object address size

	eComState := IDLE;
	
	
IDLE:	
	IF IN_bEnable THEN
		F_CreateServerHnd(	bEnable		:= FALSE,
							sSrvNetID	:= '',			// own (server) NetID
							sLocalHost	:= akuoPara.sLocalHost ,
							
							nLocalPort	:= akuoPara.iLocalPort,
							nMode		:= LISTEN_MODE_CLOSeALL OR CONNECT_MODE_ENABLEDBG, // Close all previous opened and not closed sockets and enable debug messages on socket creation/connect/close
							hServer		:= hServer );	// create server connection handle
						
		stBuffer.asduSize := F_iecApdu104ToAsduLen(fbProtocol.protPara.APDULength);
		eComState := CONNECT;
	END_IF

	
CONNECT: 
	fbConnection( 	bEnable := IN_bEnable,
					hServer	:= hServer );		
			
	CASE fbConnection.eState OF 
		eSOCKET_CONNECTED:
		
			fbProtocol.INIT( 	hSocket	:= fbConnection.hSocket, // reset fbProtocol and restart data transfer
								buffer	:= stBuffer );
			eComState := DATATRANSFER;			
		eSOCKET_DISCONNECTED:
			eComState := IDLE;	
		eSOCKET_SUSPENDED:
			; // wait for connection	
	END_CASE		
		eConnState := fbConnection.eState ;

DATATRANSFER: 
	IF IN_bEnable THEN
		fbProtocol(buffer := stBuffer);
		 eDTState := fbProtocol.eDTState ;
		IF NOT fbProtocol.bError THEN
			IF fbProtocol.eDTState = eIEC870_STARTDT THEN	
				;// exchange data
			END_IF
		ELSE // error occured - log error msg. and close socket
			(*ADSLOGSTR(	ADSLOG_MSGTYPE_ERROR OR ADSLOG_MSGTYPE_LOG,		// log errors
						'IEC60870-5-104 Transport Interface error: %s',
						DWORD_TO_HEXSTR(fbProtocol.nErrID,0,TRUE)); *)
			eComState := DISCONNECT;
		END_IF
	ELSE // stop data transfer
		eComState := DISCONNECT;
	END_IF

	
DISCONNECT: 
	fbProtocol(buffer := stBuffer);	
	fbConnection(	hServer := hServer,
					bEnable := FALSE );
					
	IF fbConnection.eState = eSOCKET_DISCONNECTED 
	AND fbProtocol.eDTState = eIEC870_STOPDT THEN
		eComState := IDLE;
	END_IF
END_CASE
END_METHOD

METHOD M_Cyclic : BOOL
VAR_INPUT
END_VAR
// Data, cyclic	
//##############################################################################################################################################//	

FOR KK := 0 TO akuoPara.iAOnb DO 
	IF AODB[KK].aObj.cfg.group.30 AND AODB[KK].aObj.obj.ident.eType<>0 THEN 
		stTxAsdu :=  AODB[KK].aObj.obj ; 

		stTxAsdu.ident.eCOT		:= eIEC870_COT_CYCLIC;	// cause of transmission - spontaneous
		stTxAsdu.ident.nORG		:= sysPara.orgAddr;				// originator address
		fbBuffer.TxAddObj(	putObj := stTxAsdu,buffer := stBuffer);
		IF NOT fbBuffer.bOk THEN
			// code for buffer overflow
			RETURN; 
		END_IF
	END_IF
END_FOR
END_METHOD

METHOD M_Init : BOOL
VAR_INPUT
END_VAR

VAR

END_VAR
END_METHOD

METHOD M_PrepareAO : BOOL
VAR_INPUT
END_VAR
VAR
	bAddCPTime		: BOOL;		// IF CP56Time is attached
	bAddQDS			: BOOL;		// If QDS is in a separate BYTE 
	QDS				: BYTE;		// QDS Value ( Quality descriptor )
	IV				: BOOL;		// INvalid
	SB				: BOOL;		//
	NT				: BOOL;		// Not topical
	BL				: BOOL;		// Blocked

	bFlicker		: BOOL;		// detect if data is flickering 

END_VAR
FOR KK := 0 TO akuoPara.iAOnb DO 
	AODB[KK].aObj.obj.ident.asduAddr	:= sysPara.asduAddr;
	AODB[KK].aObj.obj.ident.eClass		:= eIEC870_Class_1;
	
	// Get value in memory space. 
	F_iecResetStream(0,AODB[KK].aObj.obj.info.stream);
	MEMCPY( destAddr := ADR(MesDword_Old[KK]) , srcAddr := memory+ULINT_TO_DWORD(AODB[KK].aObj.cfg.byteOffs) , n := nBytesRead[KK]);
	MesCmd_old[KK] := SHR(MesDword_Old[KK] , AODB[KK].aObj.cfg.bitOffs) AND Mask[KK] ;

	CASE AODB[KK].aObj.obj.ident.eType OF 
		30:	// 
			AODB[KK].aObj.obj.ident.nObj		:= 1;
			nBytesRead[KK] := 1 ; 
			Mask[KK] := 2#1 ;
			bAddCPTime := TRUE ;
			bAddQDS		:= FALSE ;

			FB_Flicker[KK](IN_VAR:= MesCmd_old[KK].0	, IN_Window := akuoPara.tFlickerWindow , IN_COUNT:= akuoPara.uFlickerNumber , OUT_bFlicker => bFlicker );

			IF bFlicker AND akuoPara.bEnableFlicker THEN 
				BL := TRUE ;
				IV := TRUE ;
				MesCmd_old[KK].0 := 0 ;	// Freeze value .
			ELSE 
				BL := FALSE ;
				IV := FALSE ;
			END_IF
			
			
		31:
			AODB[KK].aObj.obj.ident.nObj		:= 1;
			nBytesRead[KK] := 1 ; 
			Mask[KK] := 2#11;
			bAddCPTime := TRUE ;
			bAddQDS		:= FALSE ;
		36:
			AODB[KK].aObj.obj.ident.nObj		:= 1;
			nBytesRead[KK] := 4 ; 
			Mask[KK] := 16#FFFFFFFF;	
			bAddCPTime := TRUE ;
			bAddQDS		:= TRUE ;
		13:
			AODB[KK].aObj.obj.ident.nObj		:= 1;
			nBytesRead[KK] := 4 ; 
			Mask[KK] := 16#FFFFFFFF;	
			bAddCPTime := FALSE ;
			bAddQDS		:= TRUE ;
		58:
			AODB[KK].aObj.obj.ident.nObj		:= 1;
			nBytesRead[KK] := 1 ; 
			Mask[KK] := 16#1;	
			bAddCPTime := TRUE ;		
			bAddQDS		:= FALSE ;	
	
		59:
			AODB[KK].aObj.obj.ident.nObj		:= 1;
			nBytesRead[KK] := 1 ; 
			Mask[KK] := 2#11;	
			bAddCPTime := TRUE ;
			bAddQDS		:= TRUE ;
			
		63:		// C_SE_TC_1 - Short floating point . 
			AODB[KK].aObj.obj.ident.nObj		:= 1;
			nBytesRead[KK] := 4 ; 
			Mask[KK] := 16#FFFFFFFF;	
			bAddCPTime := FALSE ;	
			bAddQDS		:= TRUE ;		
		
	END_CASE
	
	// Set Quality descriptor
	QDS:= 0;
	QDS.7 :=  IV OR AODB[KK].aObj.sts.bIV_Internal; 
	QDS.6 :=  NT ;
	QDS.5 := SB ; 
	QDS.4 := BL ;
	
	IF 	bAddQDS THEN
		F_iecCopyBufferToStream(ADR(MesCmd_old[KK]),nBytesRead[KK],AODB[KK].aObj.obj.info.stream);	// copy values TO transmit stream
		F_iecCopyBufferToStream(ADR(QDS),SIZEOF(QDS),AODB[KK].aObj.obj.info.stream);	// copy values TO transmit stream
	ELSE	
		MesCmd_old[KK] :=  MesCmd_old[KK] OR QDS ;
		F_iecCopyBufferToStream(ADR(MesCmd_old[KK]),nBytesRead[KK],AODB[KK].aObj.obj.info.stream);	// copy values TO transmit stream
	END_IF

	IF 	bAddCPTime THEN 
		F_iecCopyBufferToStream(ADR(systemTime_CP56Time2a),SIZEOF(systemTime_CP56Time2a),AODB[KK].aObj.obj.info.stream);	// copy values TO transmit stream
	END_IF
END_FOR
END_METHOD

METHOD M_ReadCmd : BOOL
VAR_INPUT
END_VAR
VAR
		MesCmd					: DWORD ;	// Processed command
		TempData_bis			: DWORD ;	// Intermediate variable

		nDCO_Cmd				: BYTE;		// Temporary variable for Double Command
		nSCO_Cmd				: BYTE ;	// Temporary variable for Single Command
		nSCO_Val				: DWORD ;	// Temporary variable for Float Command
		tActTime				: T_CP56Time2a ;
		CountAO 				: BYTE  ;	// detect if wrong IOA received
END_VAR
// -----------------------------------------------------------------------------------
// process received data
REPEAT
	fbBuffer.RxRemoveObj(	getObj => stRxAsdu,
 							buffer := stBuffer);						
	IF fbBuffer.bOk THEN
		CASE stRxAsdu.ident.eType OF
			C_IC_NA_1: 
				// General Interrogation
				F_iecCopyStreamToBuffer (ADR(nQOI),SIZEOF(nQOI), stRxAsdu.info.stream); //Copy value to local varialbe
				// create general interrogation confirmation asdu
				stTxAsdu := stRXAsdu;
				stTxAsdu.ident.eCOT := eIEC870_COT_ACT_CON; // cause of transfer -> activation confirmation
				fbBuffer.TxAddObj(	putObj := stTxAsdu,
									buffer := stBuffer);
				IF NOT fbBuffer.bOk THEN
					// code for buffer overflow (send overflow response) 

					EXIT; 
				END_IF
			
				FOR KK := 0 TO akuoPara.iAOnb DO 
				
					IF AODB[KK].aObj.cfg.group.0 AND AODB[KK].aObj.obj.ident.eType<>0 THEN 
						// create first asdu (bSlaveToMaster)
						AODB[KK].aObj.obj.ident.eCOT		:= BYTE_TO_INT(nQOI);
						AODB[KK].aObj.obj.ident.nORG		:= stRxAsdu.ident.nORG;
						stTxAsdu := AODB[KK].aObj.obj ;
	
						fbBuffer.TxAddObj(	putObj:= stTxAsdu,
											buffer:= stBuffer);
						IF NOT fbBuffer.bOk THEN
							// code for buffer overflow
							EXIT;
						END_IF	
					END_IF				
				END_FOR
				
				// create general interrogation activation termination asdu
				stTxAsdu := stRxAsdu;
				stTxAsdu.ident.eCOT := eIEC870_COT_ACT_TERM;	// cause of transfer -> activation termination
				fbBuffer.TxAddObj(	putObj:= stTxAsdu,
									buffer:= stBuffer);
				IF NOT fbBuffer.bOk THEN
					// code for buffer overflow
					EXIT; 
				END_IF			
			
			C_DC_TA_1:	// Commande Double		26 -> 43 ;	27 ->44
				CountAO := 0 ; 
				FOR KK:=1 TO akuoPara.iAOnb DO 
					IF stRxAsdu.info.objAddr = AODB[KK].aObj.obj.info.objAddr AND stRxAsdu.ident.eType = AODB[KK].aObj.obj.ident.eType THEN 
						CountAO := CountAO +1 ; ;
						F_iecCopyStreamToBuffer(ADR(nDCO_Cmd),SIZEOF(nDCO_Cmd),stRxAsdu.info.stream);
						// Get value of corresponding byte .
						TempData_bis := MesDword_Old[KK] XOR SHL(MesCmd_old[KK] ,AODB[KK].aObj.cfg.bitOffs )  ; 	// We set to zero here the bits that will be replaced
						TempData_bis := SHL(nDCO_Cmd AND Mask[KK] , AODB[KK].aObj.cfg.bitOffs) OR TempData_bis ;	// We insert the new bits 
						
						IF NOT IN_Local	THEN	
							// Apply read only if not in local . 	
							MEMCPY( destAddr := memory+ULINT_TO_DWORD(AODB[KK].aObj.cfg.byteOffs) , srcAddr := ADR(TempData_bis) , n := nBytesRead[KK]);
							MesCmd := nDCO_Cmd AND Mask[KK] ;
						ELSE
							// in local overwrite the command by the former value .
							nDCO_Cmd	:= DWORD_TO_BYTE(MesCmd_old[KK])	;
						END_IF										
						
						IF nDCO_Cmd.7 THEN
							// (1)SELECT / (0) EXECUTE STATE ( not used ) 
							; // code for select bit 
						END_IF
					
						// create activation confirmation asdu
						stTxAsdu := stRxAsdu;
						stTxAsdu.info.stream.data[0] := nDCO_Cmd;	// Permet de mettre à jour que si pas en local
						stTxAsdu.ident.eCOT := eIEC870_COT_ACT_CON; //cause of transfer -> activation confirmation
						IF IN_Local THEN
							stTxAsdu.ident.bPN :=  TRUE;
						ELSE 
							stTxAsdu.ident.bPN := FALSE;
						END_IF	
						
						fbBuffer.TxAddObj(	putObj := stTxAsdu,
											buffer := stBuffer);
						IF NOT fbBuffer.bOk THEN
							// code for buffer overflow
							EXIT; 
						END_IF
						
						IF NOT nDCO_Cmd.7 AND NOT IN_Local THEN	
	
							IF NOT (MesCmd = MesCmd_old[KK] OR IN_Local) THEN
								// Gets corresponding data type.
								stTxAsdu := AODB[KK].aObj.obj ;
								FOR JJ:= 1 TO GVL_Cst.CstNbAOEntries DO 
									IF KK<>JJ AND AODB[KK].aObj.cfg.byteOffs = AODB[JJ].aObj.cfg.byteOffs AND AODB[KK].aObj.cfg.bitOffs = AODB[JJ].aObj.cfg.bitOffs THEN
										stTxAsdu := AODB[jj].aObj.obj ;
										EXIT;
									END_IF
								END_FOR
							
								stTxAsdu.ident.eCOT		:= eIEC870_COT_RETREM;	// cause of transmission - spontaneous
								stTxAsdu.ident.nORG		:= sysPara.orgAddr;				// originator address
								
								F_iecResetStream(0,stTxAsdu.info.stream);
								F_iecCopyBufferToStream(ADR(nDCO_Cmd),SIZEOF(nDCO_Cmd),stTxAsdu.info.stream);	// copy values TO transmit stream
								fbBuffer.TxAddObj(	putObj := stTxAsdu,
													buffer := stBuffer);
								IF NOT fbBuffer.bOk THEN
									// code for buffer overflow
									RETURN; 
								END_IF	
							END_IF					
						END_IF
	
						IF NOT nDCO_Cmd.7 AND NOT IN_Local THEN	
							// code for execute function
							//create command activation termination asdu
							stTxAsdu := stRxAsdu;
							stTxAsdu.ident.eCOT := eIEC870_COT_ACT_TERM; // cause of transfer -> activation termination
							IF MesCmd = MesCmd_old[KK] THEN
								stTxAsdu.ident.bPN :=  TRUE;
							ELSE 
								stTxAsdu.ident.bPN := FALSE;
							END_IF						
					
							fbBuffer.TxAddObj(	putObj := stTxAsdu,
												buffer := stBuffer);
							IF NOT fbBuffer.bOk THEN
								// code for buffer overflow
								EXIT; 
							END_IF				
						END_IF
					END_IF
				END_FOR
				
				IF CountAO = 0 THEN 
					// code for invalid object address	IOA : return command with invalid data . 
						stTxAsdu := stRxAsdu;
						IF stRxAsdu.info.objAddr = AODB[KK].aObj.obj.info.objAddr THEN
							stTxAsdu.ident.eCOT := eIEC870_COT_UNKNOWN_TYPE; // cause of transfer -> Wrong TYPE for this IoA .  
						ELSE
							stTxAsdu.ident.eCOT := eIEC870_COT_UNKNOWN_OBJECT_ADDRESS; // cause of transfer -> unknown IOA 
						END_IF
						
						stTxAsdu.ident.bPN :=  TRUE;					
						fbBuffer.TxAddObj(	putObj := stTxAsdu,
											buffer := stBuffer);
						IF NOT fbBuffer.bOk THEN
							// code for buffer overflow
							EXIT; 
						END_IF				
					EXIT;  
				END_IF
				
			C_SC_TA_1: // single command with time tag 	30-32-33
				CountAO := 0 ; 
				FOR KK:=1 TO akuoPara.iAOnb DO 
					IF stRxAsdu.info.objAddr = AODB[KK].aObj.obj.info.objAddr THEN 
						CountAO := CountAO +1 ; ;
						F_iecCopyStreamToBuffer(ADR(nSCO_Cmd),SIZEOF(nSCO_Cmd),stRxAsdu.info.stream);
						// Get value of corresponding byte .
						TempData_bis := MesDword_Old[KK] XOR SHL(MesCmd_old[KK] ,AODB[KK].aObj.cfg.bitOffs )  ; 	// We set to zero here the bits that will be replaced
						TempData_bis := SHL(nSCO_Cmd AND Mask[KK] , AODB[KK].aObj.cfg.bitOffs) OR TempData_bis ;	// We insert the new bits 
						
						IF NOT IN_Local	THEN				// Permet de mettre à jour la commande que si pas en local
				
							MEMCPY( destAddr := memory+ULINT_TO_DWORD(AODB[KK].aObj.cfg.byteOffs) , srcAddr := ADR(TempData_bis) , n := nBytesRead[KK]);
							MesCmd := nSCO_Cmd AND Mask[KK] ;
						ELSE
							// in local overwrite the command by the former value .
							nSCO_Cmd	:= DWORD_TO_BYTE(MesCmd_old[KK])	;
	
						END_IF	
						
						IF nSCO_Cmd.7 THEN
							; // code for select bit
						END_IF
						
						// create activation confirmation asdu
						stTxAsdu := stRxAsdu;
						stTxAsdu.info.stream.data[0] := nSCO_Cmd;	// Permet de mettre à jour que si pas en local
						stTxAsdu.ident.eCOT := eIEC870_COT_ACT_CON; //cause of transfer -> activation confirmation
						
						IF IN_Local THEN
							stTxAsdu.ident.bPN :=  TRUE;
						ELSE 
							stTxAsdu.ident.bPN := FALSE;
						END_IF						
						
						fbBuffer.TxAddObj(	putObj := stTxAsdu,
											buffer := stBuffer);
						IF NOT fbBuffer.bOk THEN
							// code for buffer overflow
							EXIT; 
						END_IF
						
						
						IF NOT nSCO_Cmd.7 AND NOT IN_Local THEN
							stTxAsdu := stRxAsdu;
							stTxAsdu.ident.eCOT := eIEC870_COT_ACT_TERM; // cause of transfer -> activation termination
							stTxAsdu.ident.bPN := FALSE;
							fbBuffer.TxAddObj(	putObj := stTxAsdu,
												buffer := stBuffer);
							IF NOT fbBuffer.bOk THEN
								// code for buffer overflow
								EXIT; 
							END_IF				
						END_IF
							
					END_IF
				END_FOR
				
				IF CountAO = 0 THEN 
				// code for invalid object address	IOA : return command with invalid data . 
					stTxAsdu := stRxAsdu;
					IF stRxAsdu.info.objAddr = AODB[KK].aObj.obj.info.objAddr THEN
						stTxAsdu.ident.eCOT := eIEC870_COT_UNKNOWN_TYPE; // cause of transfer -> Wrong TYPE for this IoA .  
					ELSE
						stTxAsdu.ident.eCOT := eIEC870_COT_UNKNOWN_OBJECT_ADDRESS; // cause of transfer -> unknown IOA 
					END_IF
					stTxAsdu.ident.bPN :=  TRUE;					
					fbBuffer.TxAddObj(	putObj := stTxAsdu,
										buffer := stBuffer);
					IF NOT fbBuffer.bOk THEN
						// code for buffer overflow
						EXIT; 
					END_IF		 
					EXIT;
				END_IF
				
				
			C_SE_TC_1: // Télévaleurs	
				CountAO := 0 ; 
				FOR KK:=1 TO akuoPara.iAOnb DO 
					IF stRxAsdu.info.objAddr = AODB[KK].aObj.obj.info.objAddr THEN 
						CountAO := CountAO +1 ; ;
						F_iecCopyStreamToBuffer(ADR(nSCO_Val),SIZEOF(nSCO_Val),stRxAsdu.info.stream);
						// Get value of corresponding byte .
						TempData_bis := MesDword_Old[KK] XOR SHL(MesCmd_old[KK] ,AODB[KK].aObj.cfg.bitOffs )  ; 	// We set to zero here the bits that will be replaced
						TempData_bis := SHL(nSCO_Val AND Mask[KK] , AODB[KK].aObj.cfg.bitOffs) OR TempData_bis ;	// We insert the new bits 
			
						IF NOT IN_Local	THEN				// Permet de mettre à jour la commande que si pas en local
							MEMCPY( destAddr := memory+ULINT_TO_DWORD(AODB[KK].aObj.cfg.byteOffs) , srcAddr := ADR(TempData_bis) , n := nBytesRead[KK]);
							MesCmd := nSCO_Val AND Mask[KK] ;
					
						ELSE
							nSCO_Val := MesCmd_old[KK] ;
						END_IF	
					
						// create activation confirmation asdu
						stTxAsdu := stRxAsdu;
						F_iecCopyStreamToBufferByOffset(ADR(nSCO_Val),SIZEOF(nSCO_Val),0,stTxAsdu.info.stream);// Permet de mettre à jour que si pas en local	
						stTxAsdu.ident.eCOT := eIEC870_COT_ACT_CON; 				//cause of transfer -> activation confirmation
						
						IF IN_Local THEN
							stTxAsdu.ident.bPN :=  TRUE;
						ELSE 
							stTxAsdu.ident.bPN := FALSE;
						END_IF						
						
						fbBuffer.TxAddObj(	putObj := stTxAsdu,	buffer := stBuffer);
						IF NOT fbBuffer.bOk THEN
							// code for buffer overflow
							EXIT; 
						END_IF
						
						IF NOT IN_Local THEN
							stTxAsdu := stRxAsdu;
							stTxAsdu.ident.eCOT := eIEC870_COT_ACT_TERM; // cause of transfer -> activation termination
							stTxAsdu.ident.bPN := FALSE;
							fbBuffer.TxAddObj(	putObj := stTxAsdu,	buffer := stBuffer);
							IF NOT fbBuffer.bOk THEN
								// code for buffer overflow
								EXIT; 
							END_IF				
						END_IF
						
					END_IF
				END_FOR
				
				IF CountAO = 0 THEN 
				// code for invalid object address	IOA : return command with invalid data . 
					stTxAsdu := stRxAsdu;
					IF stRxAsdu.info.objAddr = AODB[KK].aObj.obj.info.objAddr THEN
						stTxAsdu.ident.eCOT := eIEC870_COT_UNKNOWN_TYPE; // cause of transfer -> Wrong TYPE for this IoA .  
					ELSE
						stTxAsdu.ident.eCOT := eIEC870_COT_UNKNOWN_OBJECT_ADDRESS; // cause of transfer -> unknown IOA 
					END_IF
					stTxAsdu.ident.bPN :=  TRUE;					
					fbBuffer.TxAddObj(	putObj := stTxAsdu,
										buffer := stBuffer);
					IF NOT fbBuffer.bOk THEN
						// code for buffer overflow
						EXIT; 
					END_IF		 
					EXIT;
				END_IF
			
			C_CS_NA_1: 
				// clock synchronisation
				F_iecCopyStreamToBuffer(ADR(tActTime),SIZEOF(tActTime),stRxAsdu.info.stream);	
	
				// create clock sync confirmation asdu
				stTxAsdu := stRXAsdu;
				stTxAsdu.ident.eCOT := eIEC870_COT_ACT_CON; // cause of transfer -> activation confirmation
				fbBuffer.TxAddObj(	putObj := stTxAsdu,
									buffer := stBuffer);
				IF NOT fbBuffer.bOk THEN
					// code for buffer overflow
					EXIT; 
				END_IF
				// set local computer time
				fbsetLocalTime( START	:= TRUE,
								NETID	:= '', 
								TIMESTR	:= CP56Time2a_TO_SYSTEMTIME(tActTime,20) );
				fbsetLocalTime( START	:= FALSE);
		ELSE
				// code for invalid asdu types 
				stTxAsdu := stRxAsdu;
				stTxAsdu.ident.eCOT := eIEC870_COT_UNKNOWN_TYPE; // cause of transfer -> unknown Type ASDU 
				stTxAsdu.ident.bPN :=  TRUE;					
				fbBuffer.TxAddObj(	putObj := stTxAsdu,
									buffer := stBuffer);
				IF NOT fbBuffer.bOk THEN
					// code for buffer overflow
					EXIT; 
				END_IF		
			
			EXIT;
		END_CASE
	END_IF

UNTIL NOT fbBuffer.bOk // RX fifo is empty
END_REPEAT
END_METHOD

END_FUNCTION_BLOCK

// ---- 00_FunctionsBlocks/Communication/Mail/FUN_SendMail.TcPOU
PROGRAM FUN_SendMail
////////////////// 
// Send Alarms by mails. 
//////////////////

